TYPE "C501_VAR_TME_TYPIC"
   STRUCT
      MWA { ExternalAccessible := 'False'; ExternalVisible := 'False'; ExternalWritable := 'False'} : USInt;   // Meetwaarde
      OBS { ExternalAccessible := 'False'; ExternalVisible := 'False'; ExternalWritable := 'False'} : USInt;   // Observeerbaarheid
   END_STRUCT;
END_TYPE

TYPE "C501_VAR_TRA_TYPIC"
   STRUCT
      OBS { ExternalAccessible := 'False'; ExternalVisible := 'False'; ExternalWritable := 'False'} : USInt;   // Observeerbaarheid
   END_STRUCT;
END_TYPE

TYPE "C904_STU_IF_DEB_TYPIC"
   STRUCT
      DEB_MWA { ExternalAccessible := 'False'; ExternalVisible := 'False'; ExternalWritable := 'False'} : Real;   // Meetwaarde
      EXT_AUT { ExternalAccessible := 'False'; ExternalVisible := 'False'; ExternalWritable := 'False'} : Bool;   // Externe (hoofd) beveiliging aangesproken
      EXT_HW { ExternalAccessible := 'False'; ExternalVisible := 'False'; ExternalWritable := 'False'} : Bool;   // Sturings hardware (PLC) in storing
      STO { ExternalAccessible := 'False'; ExternalVisible := 'False'; ExternalWritable := 'False'} : Struct   // Opsomming van alle storingen
         "a" : Bool;
      END_STRUCT;
   END_STRUCT;
END_TYPE

TYPE "C904_STU_IF_NIV_TYPIC"
   STRUCT
      NIV_MWA { ExternalAccessible := 'False'; ExternalVisible := 'False'; ExternalWritable := 'False'} : Real;   // Meetwaarde
      LW { ExternalAccessible := 'False'; ExternalVisible := 'False'; ExternalWritable := 'False'} : USInt;   // Stoppeil alle pompen
      SW { ExternalAccessible := 'False'; ExternalVisible := 'False'; ExternalWritable := 'False'} : USInt;   // Startpeil pomp 1 in regime leeghouden en lozen
      MSW { ExternalAccessible := 'False'; ExternalVisible := 'False'; ExternalWritable := 'False'} : USInt;   // Startpeil pomp 2 in regime leeghouden
      LHW { ExternalAccessible := 'False'; ExternalVisible := 'False'; ExternalWritable := 'False'} : USInt;   // Stoppeil bij regime Bergen
      HHW { ExternalAccessible := 'False'; ExternalVisible := 'False'; ExternalWritable := 'False'} : USInt;   // startpeil alle pompen bij regime Bergen
      EXT_AUT { ExternalAccessible := 'False'; ExternalVisible := 'False'; ExternalWritable := 'False'} : Bool;   // Externe (hoofd) beveiliging aangesproken
      EXT_HW { ExternalAccessible := 'False'; ExternalVisible := 'False'; ExternalWritable := 'False'} : Bool;   // Sturings hardware (PLC) in storing
      STO { ExternalAccessible := 'False'; ExternalVisible := 'False'; ExternalWritable := 'False'} : Struct   // Opsomming van alle storingen
         "a" : Bool;
      END_STRUCT;
   END_STRUCT;
END_TYPE

TYPE "C904_STU_IF_PMP_TYPIC"
   STRUCT
      CMD { ExternalAccessible := 'False'; ExternalVisible := 'False'; ExternalWritable := 'False'} : Bool;   // Aansturing pomp (TRUE = AAN / FALSE = UIT)
      CMD_RES { ExternalAccessible := 'False'; ExternalVisible := 'False'; ExternalWritable := 'False'} : Bool;   // Reset van de latched storingen
   END_STRUCT;
END_TYPE

TYPE "C904_VAR_DEB_TYPIC"
   STRUCT
      MWA { ExternalAccessible := 'False'; ExternalVisible := 'False'; ExternalWritable := 'False'} : USInt;   // Meetwaarde
      OBS { ExternalAccessible := 'False'; ExternalVisible := 'False'; ExternalWritable := 'False'} : USInt;   // Observeerbaarheid
   END_STRUCT;
END_TYPE

TYPE "C904_VAR_IF_PMP_TYPIC"
   STRUCT
      STS_AAN { ExternalAccessible := 'False'; ExternalVisible := 'False'; ExternalWritable := 'False'} : Bool;   // Pomp draait
      BMO_HAND { ExternalAccessible := 'False'; ExternalVisible := 'False'; ExternalWritable := 'False'} : Bool;   // Pomp in hand geschakeld
      TYD_TOT_AAN { ExternalAccessible := 'False'; ExternalVisible := 'False'; ExternalWritable := 'False'} : LInt;   // Totaal aantal draaiuren
      TYD_TOT_AAN_UUR { ExternalAccessible := 'False'; ExternalVisible := 'False'; ExternalWritable := 'False'} : LInt;   // Totaal aantal draaiuren
      TYD_AAN { ExternalAccessible := 'False'; ExternalVisible := 'False'; ExternalWritable := 'False'} : Int;   // Aantal seconden dat pomp aangeschakeld is
      TYD_UIT { ExternalAccessible := 'False'; ExternalVisible := 'False'; ExternalWritable := 'False'} : Int;   // Aantal seconden dat pomp uitgeschakeld is
      ENE_MWA1 { ExternalAccessible := 'False'; ExternalVisible := 'False'; ExternalWritable := 'False'} : Real;   // Stroommeting fase 1
      ENE_MWA2 { ExternalAccessible := 'False'; ExternalVisible := 'False'; ExternalWritable := 'False'} : Real;   // Stroommeting fase 2
      ENE_MWA3 { ExternalAccessible := 'False'; ExternalVisible := 'False'; ExternalWritable := 'False'} : Real;   // Stroommeting fase 3
      EXT_AUT { ExternalAccessible := 'False'; ExternalVisible := 'False'; ExternalWritable := 'False'} : Bool;   // Externe (hoofd) beveiliging aangesproken
      EXT_HW { ExternalAccessible := 'False'; ExternalVisible := 'False'; ExternalWritable := 'False'} : Bool;   // Sturings hardware (PLC) in storing
      STO { ExternalAccessible := 'False'; ExternalVisible := 'False'; ExternalWritable := 'False'} : Struct   // Opsomming van alle storingen
         A001 : Bool;   // Beveiliging aangesproken
         A002 : Bool;   // Storing van de motorbeveiliging van de pomp
         A003 : Bool;   // Storing motorlade
         A004 : Bool;   // Te hoge temperatuur in de motorwikkelingen
         A005 : Bool;   // Fout stroommeting fase 1
         A006 : Bool;   // Fout stroommeting fase 2
         A007 : Bool;   // Fout stroommeting fase 3
         A008 : Bool;   // Droogloop beveiliging actief: LLW vlotter bovenwater
         A009 : Bool;   // Lekdetectie pomp
         A010 : Bool;   // Motorlade uitgeschakeld
         A011 : Bool;   // Motorlade in test
         A012 : Bool;   // Motorlade uitgereden
         AT01 : Bool;   // Discordantie motor: terugmelding niet ontvangen
         AT02 : Bool;   // Discordantie motor: terugmelding blijft aanwezig
         M001 : Bool;   // Werkschakelaar uitgeschakeld
         M002 : Bool;   // Melding: Pomp heeft te lang niet gedraaid. Periodiek onderhoud nodig
      END_STRUCT;
   END_STRUCT;
END_TYPE

TYPE "C904_VAR_IF_SPI_TYPIC"
   STRUCT
      WRE { ExternalAccessible := 'False'; ExternalVisible := 'False'; ExternalWritable := 'False'} : USInt;   // Actueel actief regime
      BMO_HAND { ExternalAccessible := 'False'; ExternalVisible := 'False'; ExternalWritable := 'False'} : Bool;   // TRUE = Regime handmatig ingesteld via lokale bediening
      STO { ExternalAccessible := 'False'; ExternalVisible := 'False'; ExternalWritable := 'False'} : Struct   // Opsomming van alle storingen
         A001 : Bool;   // Beveiliging aangesproken
         A002 : Bool;   // Beveiliging No-Break aangesproken
         A003 : Bool;   // Overspanningsbeveiliging aangesproken
         A004 : Bool;   // Schuif ALSB uitgeschakeld
         A005 : Bool;   // Schuif ALSB in test
         A006 : Bool;   // Schuif ALSB uitgereden
         A007 : Bool;   // Nisdeur niet gesloten
         A008 : Bool;   // Storing tracing
      END_STRUCT;
   END_STRUCT;
END_TYPE

TYPE "C904_VAR_IF_VPI_TYPIC"
   STRUCT
      WRE { ExternalAccessible := 'False'; ExternalVisible := 'False'; ExternalWritable := 'False'} : USInt;   // Actueel actief regime
      BMO_HAND { ExternalAccessible := 'False'; ExternalVisible := 'False'; ExternalWritable := 'False'} : Bool;   // TRUE = Regime handmatig ingesteld via lokale bediening
   END_STRUCT;
END_TYPE

TYPE "C904_VAR_NIV_TYPIC"
   STRUCT
      MWA { ExternalAccessible := 'False'; ExternalVisible := 'False'; ExternalWritable := 'False'} : USInt;   // Meetwaarde
      STS_LW { ExternalAccessible := 'False'; ExternalVisible := 'False'; ExternalWritable := 'False'} : USInt;   // Stoppeil alle pompen
      STS_SW { ExternalAccessible := 'False'; ExternalVisible := 'False'; ExternalWritable := 'False'} : USInt;   // Startpeil pomp 1 in regime leeghouden en lozen
      STS_MSW { ExternalAccessible := 'False'; ExternalVisible := 'False'; ExternalWritable := 'False'} : USInt;   // Startpeil pomp 2 in regime leeghouden
      STS_LHW { ExternalAccessible := 'False'; ExternalVisible := 'False'; ExternalWritable := 'False'} : USInt;   // Stoppeil bij regime Bergen
      STS_HHW { ExternalAccessible := 'False'; ExternalVisible := 'False'; ExternalWritable := 'False'} : USInt;   // Startpeil alle pompen bij regime Bergen
      OBS { ExternalAccessible := 'False'; ExternalVisible := 'False'; ExternalWritable := 'False'} : USInt;   // Observeerbaarheid
   END_STRUCT;
END_TYPE

TYPE "C904_VAR_PMP_TYPIC"
   STRUCT
      STS { ExternalAccessible := 'False'; ExternalVisible := 'False'; ExternalWritable := 'False'} : USInt;   // Status van de pomp
      BMO { ExternalAccessible := 'False'; ExternalVisible := 'False'; ExternalWritable := 'False'} : USInt;   // Bedieningsmode
      BST { ExternalAccessible := 'False'; ExternalVisible := 'False'; ExternalWritable := 'False'} : USInt;   // Bestuurbaarheid
      LLW { ExternalAccessible := 'False'; ExternalVisible := 'False'; ExternalWritable := 'False'} : USInt;   // Vlotter droogloopbewaking
      PWR { ExternalAccessible := 'False'; ExternalVisible := 'False'; ExternalWritable := 'False'} : Real;   // Actueel vermogen van de pomp
      TYD_TOT_AAN { ExternalAccessible := 'False'; ExternalVisible := 'False'; ExternalWritable := 'False'} : USInt;   // Totaal aantal draaiuren
      TYD_AAN { ExternalAccessible := 'False'; ExternalVisible := 'False'; ExternalWritable := 'False'} : USInt;   // Tijdsduur dat pomp aangeschakeld is
      TYD_UIT { ExternalAccessible := 'False'; ExternalVisible := 'False'; ExternalWritable := 'False'} : USInt;   // Tijdsduur dat pomp uitgeschakeld is
   END_STRUCT;
END_TYPE

TYPE "C215_STU_IF_DVLU_TYPIC"
   STRUCT
      CMD_OPL { ExternalAccessible := 'False'; ExternalVisible := 'False'; ExternalWritable := 'False'} : Bool;   // Aansturing indicatiebord vluchtroute oplopende richting
      CMD_AFL { ExternalAccessible := 'False'; ExternalVisible := 'False'; ExternalWritable := 'False'} : Bool;   // Aansturing indicatiebord vluchtroute aflopende richting
      CMD_RES { ExternalAccessible := 'False'; ExternalVisible := 'False'; ExternalWritable := 'False'} : Bool;   // Reset van de latched storingen
   END_STRUCT;
END_TYPE

TYPE "C215_STU_IF_SVLU_TYPIC"
   STRUCT
      CMD_AAN { ExternalAccessible := 'False'; ExternalVisible := 'False'; ExternalWritable := 'False'} : Bool;   // Aansturing statisch indicatiebord vluchtroute
      CMD_RES { ExternalAccessible := 'False'; ExternalVisible := 'False'; ExternalWritable := 'False'} : Bool;   // Reset van de latched storingen
   END_STRUCT;
END_TYPE

TYPE "C215_VAR_DVLU_TYPIC"
   STRUCT
      STS { ExternalAccessible := 'False'; ExternalVisible := 'False'; ExternalWritable := 'False'} : USInt;   // Status van het dynamisch indicatiebord vluchtroute
      BST { ExternalAccessible := 'False'; ExternalVisible := 'False'; ExternalWritable := 'False'} : USInt;   // Bestuurbaarheid
   END_STRUCT;
END_TYPE

TYPE "C215_VAR_IF_DVLU_TYPIC"
   STRUCT
      STS_OPL { ExternalAccessible := 'False'; ExternalVisible := 'False'; ExternalWritable := 'False'} : Bool;   // Indicatiebord vluchtroute aangestuurd in oplopende richting
      STS_AFL { ExternalAccessible := 'False'; ExternalVisible := 'False'; ExternalWritable := 'False'} : Bool;   // Indicatiebord vluchtroute aangestuurd in aflopende richting
      EXT_AUT { ExternalAccessible := 'False'; ExternalVisible := 'False'; ExternalWritable := 'False'} : Bool;   // Externe (hoofd) beveiliging aangesproken
      EXT_HW { ExternalAccessible := 'False'; ExternalVisible := 'False'; ExternalWritable := 'False'} : Bool;   // Sturings hardware (PLC) in storing
      STO { ExternalAccessible := 'False'; ExternalVisible := 'False'; ExternalWritable := 'False'} : Struct   // Opsomming van alle storingen
         A001 : Bool;   // Beveiliging aangesproken
         AT01 : Bool;   // Foute terugmelding: Indicatiebord uitgestuurd, terugmelding Uit niet (of te laat) ontvangen
         AT02 : Bool;   // Foute terugmelding: Indicatiebord niet uitgestuurd, terugmelding Uit blijft aanwezig
         AT03 : Bool;   // Foute terugmelding: Oplopend aangestuurd, terugmelding Aan niet (of te laat) ontvangen
         AT04 : Bool;   // Foute terugmelding: Oplopend niet aangestuurd, terugmelding Aan blijft aanwezig
         AT05 : Bool;   // Foute terugmelding: Aflopend aangestuurd, terugmelding Aan niet (of te laat) ontvangen
         AT06 : Bool;   // Foute terugmelding: Aflopend niet aangestuurd, terugmelding Aan blijft aanwezig
         AT07 : Bool;   // Foute terugmeldingen: terugmeldingen oplopend en aflopend tegelijkertijd
      END_STRUCT;
   END_STRUCT;
END_TYPE

TYPE "C215_VAR_IF_PBK_TYPIC"
   STRUCT
      EXT_AUT { ExternalAccessible := 'False'; ExternalVisible := 'False'; ExternalWritable := 'False'} : Bool;   // Externe (hoofd) beveiliging aangesproken
      EXT_HW { ExternalAccessible := 'False'; ExternalVisible := 'False'; ExternalWritable := 'False'} : Bool;   // Sturings hardware (PLC) in storing
      STO { ExternalAccessible := 'False'; ExternalVisible := 'False'; ExternalWritable := 'False'} : Struct   // Opsomming van alle storingen
         A001 : Bool;   // Beveiliging aangesproken
         A002 : Bool;   // Storing batterij
      END_STRUCT;
   END_STRUCT;
END_TYPE

TYPE "C215_VAR_IF_SVLU_TYPIC"
   STRUCT
      STS_UIT { ExternalAccessible := 'False'; ExternalVisible := 'False'; ExternalWritable := 'False'} : Bool;   // Statisch indicatiebord vluchtroute uit
      EXT_AUT { ExternalAccessible := 'False'; ExternalVisible := 'False'; ExternalWritable := 'False'} : Bool;   // Externe (hoofd) beveiliging aangesproken
      EXT_HW { ExternalAccessible := 'False'; ExternalVisible := 'False'; ExternalWritable := 'False'} : Bool;   // Sturings hardware (PLC) in storing
      STO { ExternalAccessible := 'False'; ExternalVisible := 'False'; ExternalWritable := 'False'} : Struct   // Opsomming van alle storingen
         A001 : Bool;   // Beveiliging aangesproken
         AT01 : Bool;   // Foute terugmelding: Indicatiebord uitgestuurd, terugmelding Uit niet (of te laat) ontvangen
         AT02 : Bool;   // Foute terugmelding: Indicatiebord niet uitgestuurd, terugmelding Uit blijft aanwezig
      END_STRUCT;
   END_STRUCT;
END_TYPE

TYPE "C215_VAR_SVLU_TYPIC"
   STRUCT
      STS { ExternalAccessible := 'False'; ExternalVisible := 'False'; ExternalWritable := 'False'} : USInt;   // Status van het statisch indicatiebord vluchtroute
      BST { ExternalAccessible := 'False'; ExternalVisible := 'False'; ExternalWritable := 'False'} : USInt;   // Bestuurbaarheid
   END_STRUCT;
END_TYPE

ORGANIZATION_BLOCK "Main"   // OB1, LAD, ProgramCycle
TITLE = "Main Program Sweep (Cycle)"
{ S7_Optimized_Access := 'TRUE' }
// stored: SetENOAutomatically false
   VAR_INPUT
      Initial_Call : Bool;   // Initial call of this OB
      Remanence : Bool;   // =True, if remanent data are available
   END_VAR
BEGIN
END_ORGANIZATION_BLOCK

FUNCTION_BLOCK "TYPIC_C701_IF_KLB"   // FB120, FBD
TITLE = TYPIC_C701_IF_KLB: Brandklep
{ S7_Optimized_Access := 'TRUE' }
AUTHOR : OCOTECH
FAMILY : Typical
NAME : C701.708
// Logisch Object Besturing: C701.708
// 
// De interne functie Brandklep verzorgt de interne besturing, bewaking en fysieke aansturing van een brandklep.
// stored: MemoryReserve 10, SetENOAutomatically false
   VAR_INPUT
      IN_KLB { ExternalAccessible := 'False'; ExternalVisible := 'False'; ExternalWritable := 'False'} : Bool;   // Status brandklep (1 = Open)
   END_VAR
   VAR_OUTPUT
      VAR_IF_KLB { ExternalAccessible := 'False'; ExternalVisible := 'False'; ExternalWritable := 'False'} : "C701_VAR_IF_KLB_TYPIC";   // Struct met alle variabelen naar bovenliggende functies
   END_VAR
   VAR
      STO { ExternalWritable := 'False'} : Struct   // Storingen
         A001 : Bool;   // Brandklep gesloten
      END_STRUCT;
      VAR { ExternalWritable := 'False'} : Struct   // Variabelen
         KLB_TOE { ExternalAccessible := 'False'; ExternalVisible := 'False'} : Bool;   // Brandklep gesloten
      END_STRUCT;
   END_VAR
BEGIN

REGION Network 1: START
END_REGION

REGION Network 2: +++ Storingen +++
   // aanmaken storingen.
END_REGION

REGION Network 3: Storing A001: Brandklep gesloten
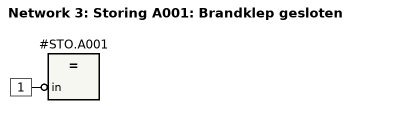
   #STO.A001 := NOT 1;
END_REGION

REGION Network 4 (SCL): EINDE
   // Variabelen van intern scada rakvlak naar outputs copieren
   #VAR_IF_KLB.KLB_TOE := #VAR.KLB_TOE;
END_REGION
END_FUNCTION_BLOCK

FUNCTION_BLOCK "TYPIC_C701_IF_KMO"   // FB102, FBD
TITLE = TYPIC_C701_IF_KMO: Koelmachine
{ S7_Optimized_Access := 'TRUE' }
AUTHOR : OCOTECH
FAMILY : Typical
NAME : C701.715
// Logisch Object Besturing: C701.715
// 
// De interne functie koelmachine verzorgt de interne besturing, bewaking en fysieke aansturing van de koelmachine behorend tot de klimaatinstallatie.
// stored: MemoryReserve 10, SetENOAutomatically false
   VAR_INPUT
      STU_IF_KMO { ExternalAccessible := 'False'; ExternalVisible := 'False'; ExternalWritable := 'False'} : Bool;   // Sturing van de interne functie klimaatregeling (IF), koudevraag voor kring
      IN_TME_IN { ExternalAccessible := 'False'; ExternalVisible := 'False'; ExternalWritable := 'False'} : Real;   // Temperatuurmeting koud water in
      IN_TME_UIT { ExternalAccessible := 'False'; ExternalVisible := 'False'; ExternalWritable := 'False'} : Real;   // Temperatuurmeting koud water uit
      IN_DME { ExternalAccessible := 'False'; ExternalVisible := 'False'; ExternalWritable := 'False'} : Real;   // Drukmeting koelen
      IN_SCF { ExternalAccessible := 'False'; ExternalVisible := 'False'; ExternalWritable := 'False'} : Bool;   // Flowmeting (1 = Flow)
      IN_FB_VGV { ExternalAccessible := 'False'; ExternalVisible := 'False'; ExternalWritable := 'False'} : Bool;   // Feedback sturing vrijgave (1 = Vrijgave)
      IN_AL { ExternalAccessible := 'False'; ExternalVisible := 'False'; ExternalWritable := 'False'} : Bool;   // Algemeen alarm koelmachine (1 = Alarm)
      IN_PMP { ExternalAccessible := 'False'; ExternalVisible := 'False'; ExternalWritable := 'False'} : Bool;   // Status circulatiepomp (1 = Aan)
      IN_AL_PMP { ExternalAccessible := 'False'; ExternalVisible := 'False'; ExternalWritable := 'False'} : Bool;   // Storing circulatiepomp (1 = Storing)
      IN_KLP { ExternalAccessible := 'False'; ExternalVisible := 'False'; ExternalWritable := 'False'} : Bool;   // Status klep (1 = Open)
   END_VAR
   VAR_OUTPUT
      VAR_IF_KMO { ExternalAccessible := 'False'; ExternalVisible := 'False'; ExternalWritable := 'False'} : "C701_VAR_IF_KMO_TYPIC";   // Struct met alle variabelen naar bovenliggende functies
      OUT_VGV { ExternalAccessible := 'False'; ExternalVisible := 'False'; ExternalWritable := 'False'} : Bool;   // Vrijgave koelmachine
      OUT_SWA_TME { ExternalAccessible := 'False'; ExternalVisible := 'False'; ExternalWritable := 'False'} : Real;   // Setpunt temperatuur koelwater
      OUT_KLP { ExternalAccessible := 'False'; ExternalVisible := 'False'; ExternalWritable := 'False'} : Bool;   // Aansturing 2wegklep
   END_VAR
   VAR
      STO { ExternalWritable := 'False'} : Struct   // Storingen
         A001 : Bool;   // Fout temperatuurmeting koelwater in
         A002 : Bool;   // Fout temperatuurmeting koelwater uit
         A003 : Bool;   // Fout drukmeting koelwater
         A004 : Bool;   // Fout flowmeting koelwater
         A005 : Bool;   // Fout algemeen koelmachine
         A006 : Bool;   // Fout circulatiepomp
      END_STRUCT;
      VAR { ExternalWritable := 'False'} : Struct   // Variabelen
         TME_IN : Real;   // Temperatuurmeting koelwater in
         TME_UIT : Real;   // Temperatuurmeting koelwater uit
         DME : Real;   // Drukmeting koelwater
         SWA_TME : Real;   // Setpunt koelwater
      END_STRUCT;
   END_VAR
BEGIN

REGION Network 1: START
END_REGION

REGION Network 2: +++ Metingen +++
   // inlezen van temperaturen en druk.
END_REGION

REGION Network 3: +++ Storingen en meldingen +++
   // aanmaken van storingen en meldingen.
END_REGION

REGION Network 4: Storing A001: Fout temperatuurmeting koelwater in
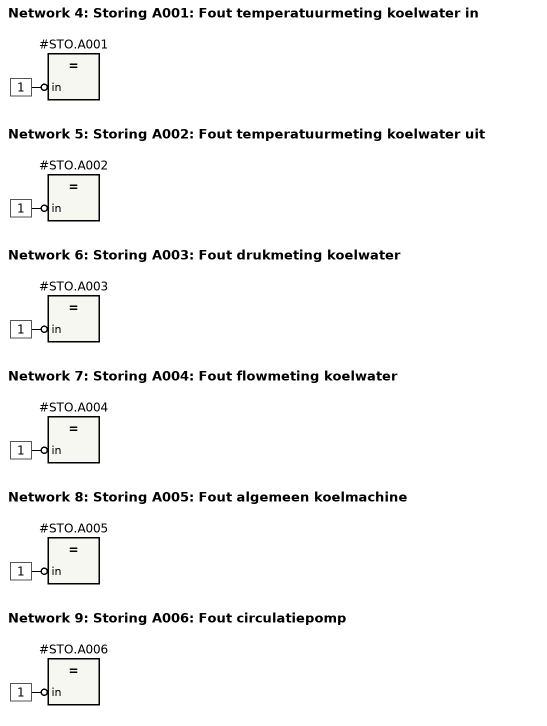
   #STO.A001 := NOT 1;
END_REGION

REGION Network 5: Storing A002: Fout temperatuurmeting koelwater uit
   #STO.A002 := NOT 1;
END_REGION

REGION Network 6: Storing A003: Fout drukmeting koelwater
   #STO.A003 := NOT 1;
END_REGION

REGION Network 7: Storing A004: Fout flowmeting koelwater
   #STO.A004 := NOT 1;
END_REGION

REGION Network 8: Storing A005: Fout algemeen koelmachine
   #STO.A005 := NOT 1;
END_REGION

REGION Network 9: Storing A006: Fout circulatiepomp
   #STO.A006 := NOT 1;
END_REGION

REGION Network 10: +++ Sturingen +++
   // sturing van klep en vrijgave koelmachine in functie van koelvraag.
END_REGION

REGION Network 11 (SCL): EINDE
   // Variabelen van intern scada rakvlak naar outputs copieren
   #VAR_IF_KMO.STO := #STO;
END_REGION
END_FUNCTION_BLOCK

FUNCTION_BLOCK "TYPIC_C701_IF_KOKR"   // FB101, FBD
TITLE = TYPIC_C701_IF_KOKR: Koelkring
{ S7_Optimized_Access := 'TRUE' }
AUTHOR : OCOTECH
FAMILY : Typical
NAME : C701.712
// Logisch Object Besturing: C701.712
// 
// De interne functie Koelkring verzorgt de interne besturing, bewaking en fysieke aansturing van een kring van de collector behorend tot de klimaatinstallatie.
// Er wordt een vrijgave aan de pompen gegeven als er een koelvraag is. De drukregeling gebeurt door de pomp zelf. Antioblokkeer beveiliging is ook instelbaar op de pomp zelf.
// Indien er een tweede pomp is, wordt deze afwisselend gebruikt. Of wordt er gewisseld bij een storing van de actieve pomp.
// De collector koelkring bestaat uit 2 kringen:
//  Kring ventiloconvectoren en klimaatkasten
//  Kring koelbatterij luchtgroep
// stored: MemoryReserve 10, SetENOAutomatically false
   VAR_INPUT
      STU_IF_KOKR { ExternalAccessible := 'False'; ExternalVisible := 'False'; ExternalWritable := 'False'} : Bool;   // Sturing van de interne functie klimaatregeling (IF), koudevraag voor kring
      IN_AAN_PMP1 { ExternalAccessible := 'False'; ExternalVisible := 'False'; ExternalWritable := 'False'} : Bool;   // Terugmelding aansturing pomp 1 (1 = Aan)
      IN_AAN_PMP2 { ExternalAccessible := 'False'; ExternalVisible := 'False'; ExternalWritable := 'False'} : Bool;   // Terugmelding aansturing pomp 2 (1 = Aan)
      IN_THM_PMP1 { ExternalAccessible := 'False'; ExternalVisible := 'False'; ExternalWritable := 'False'} : Bool;   // Status thermische beveiliging (1 = OK) pomp 1
      IN_THM_PMP2 { ExternalAccessible := 'False'; ExternalVisible := 'False'; ExternalWritable := 'False'} : Bool;   // Status thermische beveiliging (1 = OK) pomp 2
      IN_DME { ExternalAccessible := 'False'; ExternalVisible := 'False'; ExternalWritable := 'False'} : Real;   // Drukmeting
      IN_TME_IN { ExternalAccessible := 'False'; ExternalVisible := 'False'; ExternalWritable := 'False'} : Real;   // Temperatuur vertrek
      IN_TME_UIT { ExternalAccessible := 'False'; ExternalVisible := 'False'; ExternalWritable := 'False'} : Real;   // Temperatuur retour
      CFG_TYD_FB { ExternalAccessible := 'False'; ExternalVisible := 'False'; ExternalWritable := 'False'} : Time;   // Vertragingstijd storing foute terugmelding
      CFG_PMP { ExternalAccessible := 'False'; ExternalVisible := 'False'; ExternalWritable := 'False'} : Bool;   // True = Kring met 2 pompen
      CFG_PMP_TYD { ExternalAccessible := 'False'; ExternalVisible := 'False'; ExternalWritable := 'False'} : Time;   // Maximale draaitijd voor wisselen pomp
   END_VAR
   VAR_OUTPUT
      VAR_IF_KOKR { ExternalAccessible := 'False'; ExternalVisible := 'False'; ExternalWritable := 'False'} : "C701_VAR_IF_KOKR_TYPIC";   // Struct met alle variabelen naar bovenliggende functies
      OUT_VGV_PMP1 { ExternalAccessible := 'False'; ExternalVisible := 'False'; ExternalWritable := 'False'} : Bool;   // Vrijgave pomp 1
      OUT_VGV_PMP2 { ExternalAccessible := 'False'; ExternalVisible := 'False'; ExternalWritable := 'False'} : Bool;   // Vrijgave pomp 2
   END_VAR
   VAR_IN_OUT
      STU_VGV_KOKR_AAN : Bool;   // Vrijgave inschakelen NIET NODIG?
   END_VAR
   VAR
      STO { ExternalWritable := 'False'} : Struct   // Storingen
         A001 : Bool;   // Storing van de motorbeveiliging van pomp 1
         A002 : Bool;   // Storing van de motorbeveiliging van pomp 2
         A003 : Bool;   // Fout temperatuurmeting vertrek
         A004 : Bool;   // Fout temperatuurmeting retour
         A005 : Bool;   // Fout drukmeting
      END_STRUCT;
      VAR { ExternalWritable := 'False'} : Struct   // Variabelen
         TME_IN : Real;   // Temperatuur vertrek
         TME_UIT : Real;   // Temperatuur retour
         DME : Real;   // Druk vertrek
         VGV_P1 : Bool;   // Vrijgave voor pomp 1
         VGV_P2 : Bool;   // Vrijgave voor pomp 2
         TYD_TOT_AAN_P1 : LInt;   // Totaal aantal draaiuren (in seconden)
         TYD_TOT_AAN_UUR_P1 : LInt;   // Totaal aantal draaiuren (in uren)
         TYD_TOT_AAN_P2 : LInt;   // Totaal aantal draaiuren (in seconden)
         TYD_TOT_AAN_UUR_P2 : LInt;   // Totaal aantal draaiuren (in uren)
         TYD_AAN_P1 : LInt;   // Aantal seconden dat pomp aangeschakeld is
         TYD_AAN_P2 : LInt;   // Aantal seconden dat pomp aangeschakeld is
      END_STRUCT;
   END_VAR
BEGIN

REGION Network 1: START
END_REGION

REGION Network 2: +++ Metingen +++
   // inlezen van vertrek- en retourtemperatuur.
END_REGION

REGION Network 3: +++ Storingen en meldingen +++
   // aanmaken van storingen en meldingen.
END_REGION

REGION Network 4: Storing A001: Storing van de motorbeveiliging van pomp 1
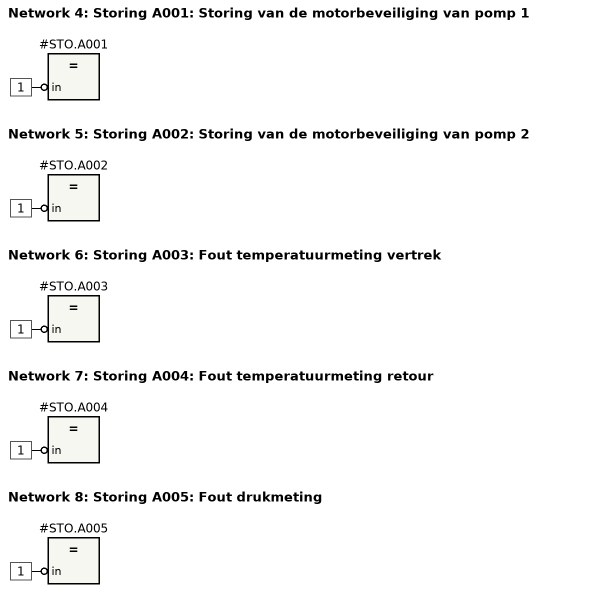
   #STO.A001 := NOT 1;
END_REGION

REGION Network 5: Storing A002: Storing van de motorbeveiliging van pomp 2
   #STO.A002 := NOT 1;
END_REGION

REGION Network 6: Storing A003: Fout temperatuurmeting vertrek
   #STO.A003 := NOT 1;
END_REGION

REGION Network 7: Storing A004: Fout temperatuurmeting retour
   #STO.A004 := NOT 1;
END_REGION

REGION Network 8: Storing A005: Fout drukmeting
   #STO.A005 := NOT 1;
END_REGION

REGION Network 9: +++ Sturingen pomp +++
   // bij koudevraag pomp vrijgave geven.
END_REGION

REGION Network 10: +++ Urentellers +++
   // tellen van de tijdsduur dat de motor draait.
END_REGION

REGION Network 11 (SCL): EINDE
   // Variabelen van intern scada rakvlak naar outputs copieren
   #VAR_IF_KOKR.STO := #STO;
END_REGION
END_FUNCTION_BLOCK

FUNCTION_BLOCK "TYPIC_C701_IF_LBS"   // FB83, FBD
TITLE = TYPIC_C701_IF_LBS: Luchtbehandelingssysteem
{ S7_Optimized_Access := 'TRUE' }
AUTHOR : OCOTECH
FAMILY : Typical
NAME : C701.702
// Logisch Object Besturing: C701.702
// 
// De interne functie Luchtbehandelingssysteem verzorgt de interne besturing, bewaking en fysieke aansturing van de luchtgroep behorend tot de klimaatinstallatie.
// stored: MemoryReserve 10, SetENOAutomatically false
   VAR_INPUT
      STU_IF_LBS_CMD { ExternalAccessible := 'False'; ExternalVisible := 'False'; ExternalWritable := 'False'} : USInt;   // Sturing van de interne functie klimaatregeling (IF), luchtgroep
      IN_DME_PU { ExternalAccessible := 'False'; ExternalVisible := 'False'; ExternalWritable := 'False'} : Real;   // Drukmeting in pulsie kanaal
      IN_DME_EX { ExternalAccessible := 'False'; ExternalVisible := 'False'; ExternalWritable := 'False'} : Real;   // Drukmeting in extractie kanaal
      IN_TME_PU { ExternalAccessible := 'False'; ExternalVisible := 'False'; ExternalWritable := 'False'} : Real;   // Temperatuurmeting in pulsie kanaal
      IN_TME_EX { ExternalAccessible := 'False'; ExternalVisible := 'False'; ExternalWritable := 'False'} : Real;   // Temperatuurmeting in extractie kanaal
      IN_TME_BU { ExternalAccessible := 'False'; ExternalVisible := 'False'; ExternalWritable := 'False'} : Real;   // Temperatuurmeting buiten
      IN_VEN_PU { ExternalAccessible := 'False'; ExternalVisible := 'False'; ExternalWritable := 'False'} : Bool;   // Status pulsie ventilator (on/off)
      IN_VEN_PU_FB { ExternalAccessible := 'False'; ExternalVisible := 'False'; ExternalWritable := 'False'} : Real;   // Feedback snelheid pulsie ventilator
      IN_VEN_PU_AUT { ExternalAccessible := 'False'; ExternalVisible := 'False'; ExternalWritable := 'False'} : Bool;   // Status thermische beveiliging pulsie ventilator (1 = OK)
      IN_VEN_PU_SCW { ExternalAccessible := 'False'; ExternalVisible := 'False'; ExternalWritable := 'False'} : Bool;   // Werkschakelaar pulsie ventilator (1 = Aan)
      IN_VEN_EX { ExternalAccessible := 'False'; ExternalVisible := 'False'; ExternalWritable := 'False'} : Bool;   // Status extractie ventilator (on/off)
      IN_VEN_EX_FB { ExternalAccessible := 'False'; ExternalVisible := 'False'; ExternalWritable := 'False'} : Real;   // Feedback snelheid extractie ventilator
      IN_VEN_EX_AUT { ExternalAccessible := 'False'; ExternalVisible := 'False'; ExternalWritable := 'False'} : Bool;   // Status thermische beveiliging extractie ventilator (1 = OK)
      IN_VEN_EX_SCW { ExternalAccessible := 'False'; ExternalVisible := 'False'; ExternalWritable := 'False'} : Bool;   // Werkschakelaar extractie ventilator (1 = Aan)
      IN_KLR_KOB { ExternalAccessible := 'False'; ExternalVisible := 'False'; ExternalWritable := 'False'} : Real;   // Feedback stand 2weg klep koelbatterij
      IN_KLR_VEB { ExternalAccessible := 'False'; ExternalVisible := 'False'; ExternalWritable := 'False'} : Real;   // Feedback stand 3weg klep verwarmingsbatterij
      IN_KLR_PU { ExternalAccessible := 'False'; ExternalVisible := 'False'; ExternalWritable := 'False'} : Real;   // Terugmelding stand open/dicht register verse lucht
      IN_KLR_EX { ExternalAccessible := 'False'; ExternalVisible := 'False'; ExternalWritable := 'False'} : Real;   // Terugmelding stand open/dicht register extractie
      IN_KLR { ExternalAccessible := 'False'; ExternalVisible := 'False'; ExternalWritable := 'False'} : Real;   // Terugmelding stand mengregister
      IN_AVR { ExternalAccessible := 'False'; ExternalVisible := 'False'; ExternalWritable := 'False'} : Bool;   // Antivries schakelaar (1 = OK)
      IN_DME_FI_VL { ExternalAccessible := 'False'; ExternalVisible := 'False'; ExternalWritable := 'False'} : Bool;   // Drukverschilmeting filter verse lucht (1 = OK)
      IN_DME_FI_EX { ExternalAccessible := 'False'; ExternalVisible := 'False'; ExternalWritable := 'False'} : Bool;   // Drukverschilmeting filter extractie (1 = OK)
      IN_WMW { ExternalAccessible := 'False'; ExternalVisible := 'False'; ExternalWritable := 'False'} : Bool;   // Terugmelding status warmtewiel (Aan / Uit)
      IN_WMW_STO { ExternalAccessible := 'False'; ExternalVisible := 'False'; ExternalWritable := 'False'} : Bool;   // Fout warmtewiel (1 = OK)
      IN_BME { ExternalAccessible := 'False'; ExternalVisible := 'False'; ExternalWritable := 'False'} : Bool;   // Rookmelder (1 = OK)
      CFG_TYD_FB { ExternalAccessible := 'False'; ExternalVisible := 'False'; ExternalWritable := 'False'} : Time;   // Vertragingstijd storing foute terugmelding
   END_VAR
   VAR_OUTPUT
      VAR_IF_LBS { ExternalAccessible := 'False'; ExternalVisible := 'False'; ExternalWritable := 'False'} : "C701_VAR_IF_LBS_TYPIC";   // Struct met alle variabelen naar bovenliggende functies
      OUT_VEN_PU_VGV { ExternalAccessible := 'False'; ExternalVisible := 'False'; ExternalWritable := 'False'} : Bool;   // Vrijgave pulsie ventilator
      OUT_VEN_PU_SNE { ExternalAccessible := 'False'; ExternalVisible := 'False'; ExternalWritable := 'False'} : Real;   // Snelheid pulsie ventilator
      OUT_VEN_EX_VGV { ExternalAccessible := 'False'; ExternalVisible := 'False'; ExternalWritable := 'False'} : Bool;   // Vrijgave extractie ventilator
      OUT_VEN_EX_SNE { ExternalAccessible := 'False'; ExternalVisible := 'False'; ExternalWritable := 'False'} : Real;   // Snelheid extractie ventilator
      OUT_KLR_KOB { ExternalAccessible := 'False'; ExternalVisible := 'False'; ExternalWritable := 'False'} : Real;   // Aansturing klep koelbatterij
      OUT_KLR_VEB { ExternalAccessible := 'False'; ExternalVisible := 'False'; ExternalWritable := 'False'} : Real;   // Aansturing klep verwarmingsbatterij
      OUT_KLR_VL { ExternalAccessible := 'False'; ExternalVisible := 'False'; ExternalWritable := 'False'} : Real;   // Damper verse lucht sturing
      OUT_KLR_EX { ExternalAccessible := 'False'; ExternalVisible := 'False'; ExternalWritable := 'False'} : Real;   // Damper extractie lucht sturing
      OUT_KLR { ExternalAccessible := 'False'; ExternalVisible := 'False'; ExternalWritable := 'False'} : Real;   // Aansturing positie mengregister
      OUT_WMW { ExternalAccessible := 'False'; ExternalVisible := 'False'; ExternalWritable := 'False'} : Real;   // Aansturing recuperatie warmtewisselaar
   END_VAR
   VAR_IN_OUT
      STU_VGV_PMP_AAN : Bool;   // Vrijgave inschakelen
   END_VAR
   VAR
      BED : Struct   // Bedieningen
         REM : Bool;   // Bediening om luchtgroep in remote te schakelen
         NORMAAL : Bool;   // Bediening om luchtgroep in regime Normaal te schakelen
         RECIRCULATIE : Bool;   // Bediening om luchtgroep in regime Recirculatie te schakelen
         UIT : Bool;   // Bediening om luchtgroep in regime Uit te schakelen
      END_STRUCT;
      STO { ExternalWritable := 'False'} : Struct   // Storingen
         A001 : Bool;   // Storing van de motorbeveiliging van pulsie ventilator
         A002 : Bool;   // Storing van de motorbeveiliging van extractie ventilator
         A003 : Bool;   // Fout drukmeting pulsie
         A004 : Bool;   // Fout drukmeting extractie
         A005 : Bool;   // Fout temperatuurmeting pulsie
         A006 : Bool;   // Fout temperatuurmeting extractie
         A007 : Bool;   // Fout temperatuurmeting buitenlucht
         A008 : Bool;   // Antivries alarm
         A009 : Bool;   // Filter vuil verse lucht
         A010 : Bool;   // Filter vuil extractie lucht
         AT01 : Bool;   // Foute terugmelding: damper verse lucht aangestuurd, terugmelding niet (of te laat) ontvangen
         AT02 : Bool;   // Foute terugmelding: damper extractie lucht aangestuurd, terugmelding niet (of te laat) ontvangen
         M001 : Bool;   // De pulsie ventilator is afgekoppeld via de werkschakelaar
         M002 : Bool;   // De extractie ventilator is afgekoppeld via de werkschakelaar
      END_STRUCT;
      VAR { ExternalWritable := 'False'} : Struct   // Variabelen
         PID_P_PU : Real;   // P factor van PID regeling voor pulsie ventilator
         PID_I_PU : Time;   // Integratietijd van PID regeling voor pulsie ventilator
         PID_D_PU : Time;   // D actie van PID regeling voor pulsie ventilator
         PID_P_EX : Real;   // P factor van PID regeling voor extractie ventilator
         PID_I_EX : Time;   // Integratietijd van PID regeling voor extractie ventilator
         PID_D_EX : Time;   // D actie van PID regeling voor extractie ventilator
         PID_P_KOB : Real;   // P factor van PID regeling voor klep van koelbatterij
         PID_I_KOB : Time;   // Integratietijd van PID regeling voor klep van koelbatterij
         PID_D_KOB : Time;   // D actie van PID regeling voor klep van koelbatterij
         PID_P_VEB : Real;   // P factor van PID regeling voor klep van verwarmingsbatterij
         PID_I_VEB : Time;   // Integratietijd van PID regeling voor klep van verwarmingsbatterij
         PID_D_VEB : Time;   // D actie van PID regeling voor klep van verwarmingsbatterij
         SWA_D_PU : Real;   // Setpunt druk pulsie kanaal
         SWA_D_EX : Real;   // Setpunt druk extractie kanaal
         SWA_T_PU : Real;   // Setpunt temperatuur pulsie
         DME_PU : Real;   // Drukmeting pulsie kanaal
         DME_EX : Real;   // Drukmeting extractie kanaal
         TME_PU : Real;   // Temperatuurmeting in pulsie
         TME_EX : Real;   // Temperatuurmeting in extractie
         TME_BU : Real;   // Temperatuurmeting buitenlucht
         WRE { ExternalAccessible := 'False'; ExternalVisible := 'False'} : USInt;   // Werkingsregime
         BMO_HAND { ExternalAccessible := 'False'; ExternalVisible := 'False'} : Bool;   // TRUE = Werkingsregime is handmatig ingesteld via lokale bediening
         "Vrijgave pomp verwarmingsbat" { ExternalAccessible := 'False'; ExternalVisible := 'False'} : Bool;   // Gaat naar if verwarmingskring CHECKEN OF DEZE POMP NU HIER INZIT OF IN DE KRING
         REQ_VE { ExternalAccessible := 'False'; ExternalVisible := 'False'} : Bool;   // Warmtevraag voor kring verwarmingsbatterijen
         REQ_KO { ExternalAccessible := 'False'; ExternalVisible := 'False'} : Bool;   // Koelvraag voor kring koelbatterijen (luchtgroep)
      END_STRUCT;
   END_VAR
BEGIN

REGION Network 1: START
END_REGION

REGION Network 2: +++ Metingen +++
   // inlezen van de temperatuur en drukken.
END_REGION

REGION Network 3: +++ Storingen en meldingen +++
   // aanmaken van de storingen en meldingen.
END_REGION

REGION Network 4: Storing A001: Storing van de motorbeveiliging van pulsie ventilator
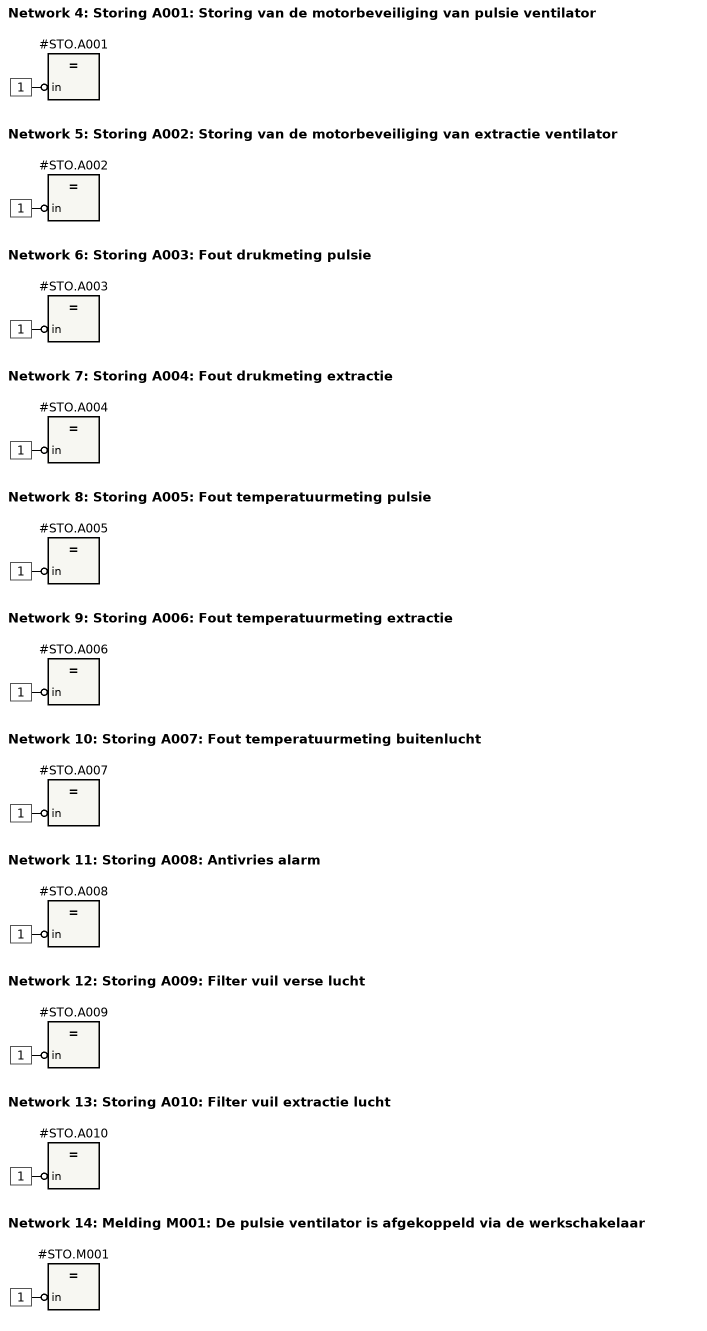
   #STO.A001 := NOT 1;
END_REGION

REGION Network 5: Storing A002: Storing van de motorbeveiliging van extractie ventilator
   #STO.A002 := NOT 1;
END_REGION

REGION Network 6: Storing A003: Fout drukmeting pulsie
   #STO.A003 := NOT 1;
END_REGION

REGION Network 7: Storing A004: Fout drukmeting extractie
   #STO.A004 := NOT 1;
END_REGION

REGION Network 8: Storing A005: Fout temperatuurmeting pulsie
   #STO.A005 := NOT 1;
END_REGION

REGION Network 9: Storing A006: Fout temperatuurmeting extractie
   #STO.A006 := NOT 1;
END_REGION

REGION Network 10: Storing A007: Fout temperatuurmeting buitenlucht
   #STO.A007 := NOT 1;
END_REGION

REGION Network 11: Storing A008: Antivries alarm
   #STO.A008 := NOT 1;
END_REGION

REGION Network 12: Storing A009: Filter vuil verse lucht
   #STO.A009 := NOT 1;
END_REGION

REGION Network 13: Storing A010: Filter vuil extractie lucht
   #STO.A010 := NOT 1;
END_REGION

REGION Network 14: Melding M001: De pulsie ventilator is afgekoppeld via de werkschakelaar
   #STO.M001 := NOT 1;
END_REGION

REGION Network 15: Melding M002: De extractie ventilator is afgekoppeld via de werkschakelaar
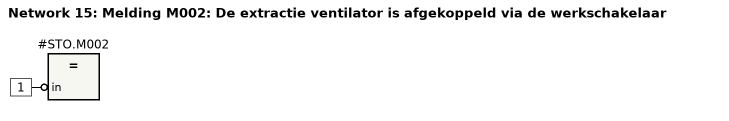
   #STO.M002 := NOT 1;
END_REGION

REGION Network 16: +++ Regelingen +++
   // PID regelingen voor luchtdebiet en temperatuur.
END_REGION

REGION Network 17: +++ Sturingen +++
   // aansturingen bepaalt door de uitgangen van de PID regelaars.
END_REGION

REGION Network 18 (SCL): EINDE
   // Variabelen van intern scada rakvlak naar outputs copieren
   #VAR_IF_LBS.WRE := #VAR.WRE;
   #VAR_IF_LBS.BMO_HAND := #VAR.BMO_HAND;
   #VAR_IF_LBS."Vrijgave pomp verwarmingsbat" := #VAR."Vrijgave pomp verwarmingsbat";
   #VAR_IF_LBS.REQ_VE := #VAR.REQ_VE;
   #VAR_IF_LBS.REQ_KO := #VAR.REQ_KO;
   #VAR_IF_LBS.STO := #STO;
END_REGION
END_FUNCTION_BLOCK

FUNCTION_BLOCK "TYPIC_C701_IF_VAT"   // FB69, FBD
TITLE = TYPIC_C701_IF_VAT: Expansievaten
{ S7_Optimized_Access := 'TRUE' }
AUTHOR : OCOTECH
FAMILY : Typical
NAME : C701.713
// Logisch Object Besturing: C701.713
// 
// De interne functie Expansievaten verzorgt de bewaking van een expansievat behorend tot de klimaatinstallatie.
// In zowel de collector verwarming als koeling is er een expansievat.
// stored: MemoryReserve 10, SetENOAutomatically false
   VAR_INPUT
      IN_AL_VE { ExternalAccessible := 'False'; ExternalVisible := 'False'; ExternalWritable := 'False'} : Bool;   // Alarm lage druk expansievat verwarming (1 = Alarm)
      IN_DME_VE { ExternalAccessible := 'False'; ExternalVisible := 'False'; ExternalWritable := 'False'} : Real;   // Drukmeting expansievat verwarming
      IN_AL_KO { ExternalAccessible := 'False'; ExternalVisible := 'False'; ExternalWritable := 'False'} : Bool;   // Alarm lage druk expansievat koeling (1 = Alarm)
      IN_DME_KO { ExternalAccessible := 'False'; ExternalVisible := 'False'; ExternalWritable := 'False'} : Real;   // Drukmeting expansievat koeling
   END_VAR
   VAR_OUTPUT
      VAR_IF_VAT { ExternalAccessible := 'False'; ExternalVisible := 'False'; ExternalWritable := 'False'} : "C701_VAR_IF_VAT_TYPIC";   // Struct met alle variabelen naar bovenliggende functies
   END_VAR
   VAR
      STO { ExternalWritable := 'False'} : Struct   // Storingen
         A001 : Bool;   // Alarm lage druk expansievat verwarming
         A002 : Bool;   // Fout drukmeting expansievat verwarming
         A003 : Bool;   // Alarm lage druk expansievat koeling
         A004 : Bool;   // Fout drukmeting expansievat koeling
      END_STRUCT;
      VAR { ExternalWritable := 'False'} : Struct   // Variabelen
         DME_VE : Real;   // Drukmeting expansievat verwarming
         DME_KO : Real;   // Drukmeting expansievat koeling
      END_STRUCT;
   END_VAR
BEGIN

REGION Network 1: START
END_REGION

REGION Network 2: +++ Metingen +++
   // inlezen van drukmeting.
END_REGION

REGION Network 3: +++ Storingen en meldingen +++
   // aanmaken van storingen en meldingen.
END_REGION

REGION Network 4: Storing A001: Alarm lage druk expansievat verwarming
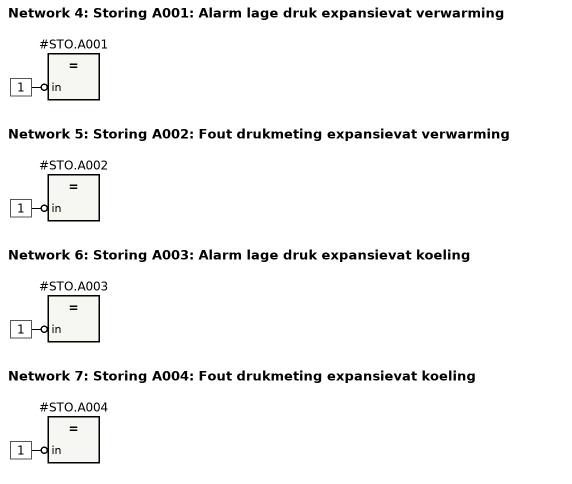
   #STO.A001 := NOT 1;
END_REGION

REGION Network 5: Storing A002: Fout drukmeting expansievat verwarming
   #STO.A002 := NOT 1;
END_REGION

REGION Network 6: Storing A003: Alarm lage druk expansievat koeling
   #STO.A003 := NOT 1;
END_REGION

REGION Network 7: Storing A004: Fout drukmeting expansievat koeling
   #STO.A004 := NOT 1;
END_REGION

REGION Network 8 (SCL): EINDE
   // Variabelen van intern scada rakvlak naar outputs copieren
   #VAR_IF_VAT.STO := #STO;
END_REGION
END_FUNCTION_BLOCK

FUNCTION_BLOCK "TYPIC_C701_IF_VAT_BUF"   // FB70, FBD
TITLE = TYPIC_C701_IF_VAT_BUF: Buffervat warm water
{ S7_Optimized_Access := 'TRUE' }
AUTHOR : OCOTECH
FAMILY : Typical
NAME : C701.714
// Logisch Object Besturing: C701.714
// 
// De interne functie Buffervat verzorgt de interne besturing, bewaking en fysieke aansturing van het buffervat behorend tot de klimaatinstallatie.
// stored: MemoryReserve 10, SetENOAutomatically false
   VAR_INPUT
      STU_IF_VAT_BUF { ExternalAccessible := 'False'; ExternalVisible := 'False'; ExternalWritable := 'False'} : Bool;   // Sturing van de interne functie klimaatregeling (IF), vrijgave door storing warmtepomp
      IN_STO { ExternalAccessible := 'False'; ExternalVisible := 'False'; ExternalWritable := 'False'} : Bool;   // Storing elektrisch weerstand
      IN_TME_MWA_INV { ExternalAccessible := 'False'; ExternalVisible := 'False'; ExternalWritable := 'False'} : Real;   // Temperatuurmeting warmwater in vertrek
      IN_TME_MWA_UITV { ExternalAccessible := 'False'; ExternalVisible := 'False'; ExternalWritable := 'False'} : Real;   // Temperatuurmeting warmwater uit vertrek
      IN_TME3_MWA { ExternalAccessible := 'False'; ExternalVisible := 'False'; ExternalWritable := 'False'} : Real;   // Temperatuurmeting warmwater in retour
      IN_TME4_MWA { ExternalAccessible := 'False'; ExternalVisible := 'False'; ExternalWritable := 'False'} : Real;   // Temperatuurmeting warmwater uit retour
   END_VAR
   VAR_OUTPUT
      VAR_IF_VAT_BUF { ExternalAccessible := 'False'; ExternalVisible := 'False'; ExternalWritable := 'False'} : "C701_VAR_IF_VAT_BUF_TYPIC";   // Struct met alle variabelen naar bovenliggende functies
      OUT_AAN { ExternalAccessible := 'False'; ExternalVisible := 'False'; ExternalWritable := 'False'} : Bool;   // Sturing elektrische weerstand (1 = Aan)
   END_VAR
   VAR
      STO { ExternalWritable := 'False'} : Struct   // Storingen
         A001 : Bool;   // Fout temperatuurmeting in vertrek
         A002 : Bool;   // Fout temperatuurmeting uit vertrek
         A003 : Bool;   // Fout temperatuurmeting in retour
         A004 : Bool;   // Fout temperatuurmeting uit retour
      END_STRUCT;
      VAR { ExternalWritable := 'False'} : Struct   // Variabelen
         TME_IN_VERTREK : Real;   // Temperatuurmeting in
         TME_UIT_VERTREK : Real;   // Temperatuurmeting uit
         TME_IN_RETOUR : Real;   // Temperatuurmeting in
         TME_UIT_RETOUR : Real;   // Temperatuurmeting uit
         TME_SWA : Real;   // Setpunt temperatuur buffervat
      END_STRUCT;
   END_VAR
BEGIN

REGION Network 1: START
END_REGION

REGION Network 2: +++ Metingen +++
   // inlezen van ingaande en uitgaande temperatuur.
END_REGION

REGION Network 3: +++ Storingen en meldingen +++
   // aanmaken van storingen en meldingen.
END_REGION

REGION Network 4: Storing A001: Fout temperatuurmeting in vertrek
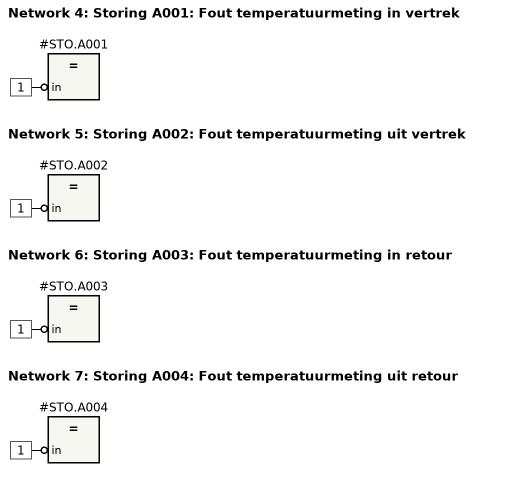
   #STO.A001 := NOT 1;
END_REGION

REGION Network 5: Storing A002: Fout temperatuurmeting uit vertrek
   #STO.A002 := NOT 1;
END_REGION

REGION Network 6: Storing A003: Fout temperatuurmeting in retour
   #STO.A003 := NOT 1;
END_REGION

REGION Network 7: Storing A004: Fout temperatuurmeting uit retour
   #STO.A004 := NOT 1;
END_REGION

REGION Network 8: +++ Sturingen +++
   // bij storing warmtepomp wordt elektrische weerstand vrijgegeven en geregeld naar setpunt.
END_REGION

REGION Network 9 (SCL): EINDE
   // Variabelen van intern scada rakvlak naar outputs copieren
   #VAR_IF_VAT_BUF.STO := #STO;
END_REGION
END_FUNCTION_BLOCK

FUNCTION_BLOCK "TYPIC_C701_IF_VEKR"   // FB96, FBD
TITLE = TYPIC_C701_IF_VEKR: Verwarmingskring
{ S7_Optimized_Access := 'TRUE' }
AUTHOR : OCOTECH
FAMILY : Typical
NAME : C701.711
// Logisch Object Besturing: C701.711
// 
// 								De interne functie Verwarmingskring verzorgt de interne besturing,
// 								bewaking en fysieke aansturing van een collectorkring behorend tot
// 								de klimaatinstallatie.
// 								Er wordt een vrijgave aan de pompen gegeven als er een warmtevraag
// 								is. De drukregeling gebeurt door de pomp zelf. Antioblokkeer
// 								beveiliging is ook instelbaar op de pomp zelf.
// 								De collector verwarming bestaat uit 2 kringen:
// 								Kring verwarmingsbatterijen
// 								Kring ventiloconvectoren en klimaatkasten
// stored: MemoryReserve 10, SetENOAutomatically false
   VAR_INPUT
      STU_IF_VEKR { ExternalAccessible := 'False'; ExternalVisible := 'False'; ExternalWritable := 'False'} : Bool;   // Sturing van de interne functie klimaatregeling (IF), warmtevraag voor kring
      IN_AAN_PMP { ExternalAccessible := 'False'; ExternalVisible := 'False'; ExternalWritable := 'False'} : Bool;   // Terugmelding aansturing pomp (1 = Aan)
      IN_THM { ExternalAccessible := 'False'; ExternalVisible := 'False'; ExternalWritable := 'False'} : Bool;   // Status thermische beveiliging (1 = OK)
      IN_DME { ExternalAccessible := 'False'; ExternalVisible := 'False'; ExternalWritable := 'False'} : Real;   // Drukmeting
      IN_TME_IN { ExternalAccessible := 'False'; ExternalVisible := 'False'; ExternalWritable := 'False'} : Real;   // Temperatuur vertrek
      IN_TME_UIT { ExternalAccessible := 'False'; ExternalVisible := 'False'; ExternalWritable := 'False'} : Real;   // Temperatuur retour
      CFG_TYD_FB { ExternalAccessible := 'False'; ExternalVisible := 'False'; ExternalWritable := 'False'} : Time;   // Vertragingstijd storing foute terugmelding
   END_VAR
   VAR_OUTPUT
      VAR_IF_VEKR { ExternalAccessible := 'False'; ExternalVisible := 'False'; ExternalWritable := 'False'} : "C701_VAR_IF_VEKR_TYPIC";   // Struct met alle variabelen naar bovenliggende functies
      OUT_VGV { ExternalAccessible := 'False'; ExternalVisible := 'False'; ExternalWritable := 'False'} : Bool;   // Vrijgave pomp
   END_VAR
   VAR_IN_OUT
      STU_VGV_VEKR_AAN : Bool;   // Vrijgave inschakelen NIET NODIG?
   END_VAR
   VAR
      STO { ExternalWritable := 'False'} : Struct   // Storingen
         A001 : Bool;   // Storing van de motorbeveiliging van de pomp
         A002 : Bool;   // Fout temperatuurmeting vertrek
         A003 : Bool;   // Fout temperatuurmeting retour
         A004 : Bool;   // Fout drukmeting
         M001 : Bool;   // De motor is afgekoppeld via de werkschakelaar
      END_STRUCT;
      VAR { ExternalWritable := 'False'} : Struct   // Variabelen
         TME_IN : Real;   // Temperatuur vertrek
         TME_UIT : Real;   // Temperatuur retour
         DME : Real;   // Druk vertrek
         VGV : Bool;   // Vrijgave voor pomp
         TYD_TOT_AAN : LInt;   // Totaal aantal draaiuren (in seconden)
         TYD_TOT_AAN_UUR : LInt;   // Totaal aantal draaiuren (in uren)
      END_STRUCT;
   END_VAR
BEGIN

REGION Network 1: START
END_REGION

REGION Network 2: +++ Metingen +++
   // inlezen van vertrek- en retourtemperatuur.
END_REGION

REGION Network 3: +++ Storingen en meldingen +++
   // aanmaken van storingen en meldingen.
END_REGION

REGION Network 4: Storing A001: Storing van de motorbeveiliging van de pomp
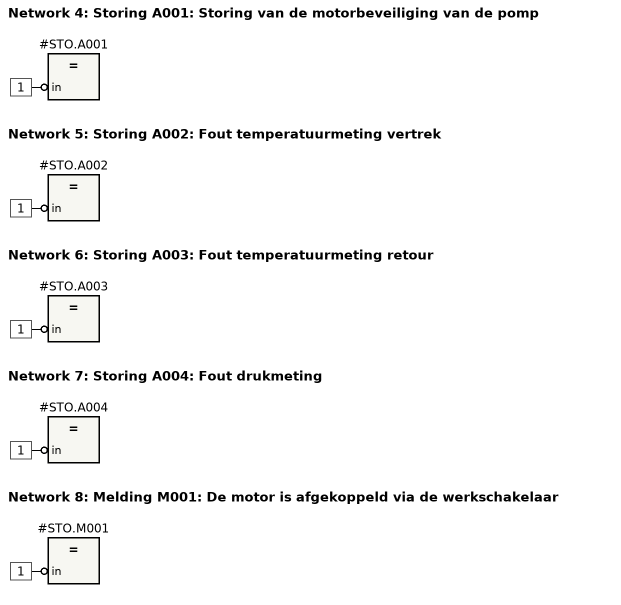
   #STO.A001 := NOT 1;
END_REGION

REGION Network 5: Storing A002: Fout temperatuurmeting vertrek
   #STO.A002 := NOT 1;
END_REGION

REGION Network 6: Storing A003: Fout temperatuurmeting retour
   #STO.A003 := NOT 1;
END_REGION

REGION Network 7: Storing A004: Fout drukmeting
   #STO.A004 := NOT 1;
END_REGION

REGION Network 8: Melding M001: De motor is afgekoppeld via de werkschakelaar
   #STO.M001 := NOT 1;
END_REGION

REGION Network 9: +++ Sturingen pomp +++
   // bij warmtevraag pomp vrijgave geven.
END_REGION

REGION Network 10: +++ Urentellers +++
   // tellen van de tijdsduur dat de motor draait.
END_REGION

REGION Network 11 (SCL): EINDE
   // Variabelen van intern scada rakvlak naar outputs copieren
   #VAR_IF_VEKR.STO := #STO;
END_REGION
END_FUNCTION_BLOCK

FUNCTION_BLOCK "TYPIC_C104_BF_NSI"   // FB95, FBD
TITLE = TYPIC_C104_BF_NSI: Noodstroominstallatie
{ S7_Optimized_Access := 'TRUE' }
AUTHOR : OCOTECH
FAMILY : Typical
NAME : C104.801
// Logisch Object Besturing: C104.801
// 
// Het doel van de BF NSI (noodstroominstallatie) is om de algemene opvolging te voorzien van de noodstroominstallatie.
// stored: MemoryReserve 10, SetENOAutomatically false
   VAR_INPUT
      STU_ALG_LCK_SIG { ExternalAccessible := 'False'; ExternalVisible := 'False'; ExternalWritable := 'False'} : USInt;   // Onderdruk alarmen
   END_VAR
   VAR_OUTPUT
      VAR_ENE_TOT_NSI { ExternalAccessible := 'False'; ExternalVisible := 'False'; ExternalWritable := 'False'} : Real;   // Totaal energieverbruik noodstroominstallatie
      VAR_VGV_NSI { ExternalAccessible := 'False'; ExternalVisible := 'False'; ExternalWritable := 'False'} : USInt;   // Vrijgave: alle noodstroomaggregaten lopen synchroon
   END_VAR
   VAR_IN_OUT
      VAR_IF_NSI : "C104_VAR_IF_NSI_TYPIC";   // Struct met alle variabelen ontvangen van de interne besturing (PMS) van de noodstroominstallatie
   END_VAR
   VAR
      SIG { ExternalWritable := 'False'} : Struct   // Signaleringen
         AB01 : Bool;   // Noodstroominstallatie niet beschikbaar
         AB02 : Bool;   // Noodstroominstallatie beperkt beschikbaar
      END_STRUCT;
      VAR { ExternalWritable := 'False'} : Struct   // Variabelen
         BSC : USInt;   // Geeft de beschikbaarheid van de noodstroominstallatie aan
         VGV_SIG_VOP : Bool;   // TRUE = Signaleringen vrijgegeven voor verkeersoperator FALSE = Onderdrukt
      END_STRUCT;
   END_VAR
BEGIN

REGION Network 1: START
END_REGION

REGION Network 2: +++ Bepalen beschikbaarheidsstatus +++
   // Beschikbaarheidsstatus (beschikbaar / beperkt beschikbaar / niet beschikbaar) bepalen.
END_REGION

REGION Network 3 (SCL): Beschikbaarheidsstatus bepalen
   IF 
       //voorwaarden "Niet beschikbaar"
       TRUE
   THEN
       //Beschikbaarheidsstatus = Niet Beschikbaar
       #VAR.BSC:= "NietBeschikbaar";
   ELSIF
       //voorwaarden "Beperkt beschikbaar"
       TRUE
   THEN
       //Beschikbaarheidsstatus = Beperkt Beschikbaar
       #VAR.BSC:= "Beperkt";
   ELSE
       //Beschikbaarheidsstatus = Beschikbaar
       #VAR.BSC:= "Beschikbaar";
   END_IF;
END_REGION

REGION Network 4: +++ Doorkoppeling totale energieverbruik HSI +++
   // Het ontvangen energieverbruik ter beschikking stellen.
END_REGION

REGION Network 5: +++ Signaleringen +++
   // Aanmaken signaleringen.
END_REGION

REGION Network 6: Signalering AB01 : Niet Beschikbaar
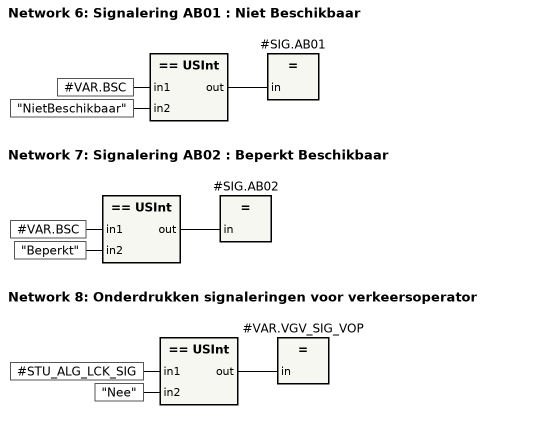
   #SIG.AB01 := #VAR.BSC = "NietBeschikbaar";
END_REGION

REGION Network 7: Signalering AB02 : Beperkt Beschikbaar
   #SIG.AB02 := #VAR.BSC = "Beperkt";
END_REGION

REGION Network 8: Onderdrukken signaleringen voor verkeersoperator
   // Via de variabele VGV_SIG_VOP wordt aan IRIS SCADA doorgegeven of signaleringen (bestemd voor de verkeersoperator) van de deze functie zichtbaar (of onderdrukt) moeten zijn.
   #VAR.VGV_SIG_VOP := #STU_ALG_LCK_SIG = "Nee";
END_REGION

REGION Network 9: EINDE
   // Variabelen van intern scada rakvlak naar outputs copieren
END_REGION
END_FUNCTION_BLOCK

FUNCTION_BLOCK "TYPIC_C104_IF_KLP"   // FB94, FBD
TITLE = TYPIC_C104_IF_KLP: Brandstofklep
{ S7_Optimized_Access := 'TRUE' }
AUTHOR : OCOTECH
FAMILY : Typical
NAME : C104.705
// Logisch Object Besturing: C104.705
// 
// De interne functie Brandstofklep verzorgt de bewaking van een brandstofklep van een noodstroomaggregaat.
// stored: MemoryReserve 10, SetENOAutomatically false
   VAR_INPUT
      EXT_AUT { ExternalAccessible := 'False'; ExternalVisible := 'False'; ExternalWritable := 'False'} : Bool;   // Externe (hoofd) beveiliging (1 = OK)
      EXT_HW { ExternalAccessible := 'False'; ExternalVisible := 'False'; ExternalWritable := 'False'} : Bool;   // Sturings hardware (PLC) bewaking (1 = OK)
      IN_STO_NOK { ExternalAccessible := 'False'; ExternalVisible := 'False'; ExternalWritable := 'False'} : Bool;   // Storing aanwezig die niet observeerbaar tot gevolg heeft
      IN_STO_OK { ExternalAccessible := 'False'; ExternalVisible := 'False'; ExternalWritable := 'False'} : Bool;   // Storing aanwezig die observeerbaarheid niet beinvloed
      IN_OPEN { ExternalAccessible := 'False'; ExternalVisible := 'False'; ExternalWritable := 'False'} : Bool;   // Brandstofklep open
      IN_TOE { ExternalAccessible := 'False'; ExternalVisible := 'False'; ExternalWritable := 'False'} : Bool;   // Brandstofklep dicht
      IN_AUT_C104 { ExternalAccessible := 'False'; ExternalVisible := 'False'; ExternalWritable := 'False'} : Bool;   // Beveiligingen: serie geschakelde terugmelding (1 = OK)
   END_VAR
   VAR_OUTPUT
      VAR_IF_KLP { ExternalAccessible := 'False'; ExternalVisible := 'False'; ExternalWritable := 'False'} : "C104_VAR_IF_KLP_TYPIC";   // Struct met alle variabelen naar bovenliggende functies
   END_VAR
   VAR
      STO { ExternalWritable := 'False'} : Struct   // Storingen
         A001 : Bool;   // Beveiliging aangesproken
         A002 : Bool;   // Brandstofklep in storing
         A003 : Bool;   // Algemene storing brandstofklep
      END_STRUCT;
      VAR { ExternalWritable := 'False'} : Struct   // Variabelen
         OPEN { ExternalAccessible := 'False'; ExternalVisible := 'False'} : Bool;   // Brandstofklep open
         TOE { ExternalAccessible := 'False'; ExternalVisible := 'False'} : Bool;   // Brandstofklep dicht
         EXT_AUT { ExternalAccessible := 'False'; ExternalVisible := 'False'} : Bool;   // Externe (hoofd) beveiliging aangesproken
         EXT_HW { ExternalAccessible := 'False'; ExternalVisible := 'False'} : Bool;   // Sturings hardware (PLC) in storing
      END_STRUCT;
   END_VAR
BEGIN

REGION Network 1: START
END_REGION

REGION Network 2: +++ Verwerking statussen +++
   // Bepalen van de statussen van de brandstofklep.
END_REGION

REGION Network 3: +++ Storingen +++
   // Verwerken van de storingsmeldingen (inputs).
END_REGION

REGION Network 4: Storing A001: Beveiliging aangesproken
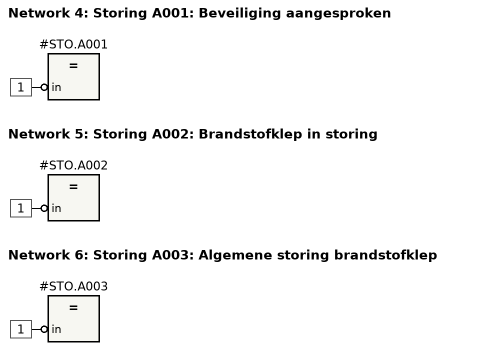
   #STO.A001 := NOT 1;
END_REGION

REGION Network 5: Storing A002: Brandstofklep in storing
   #STO.A002 := NOT 1;
END_REGION

REGION Network 6: Storing A003: Algemene storing brandstofklep
   #STO.A003 := NOT 1;
END_REGION

REGION Network 7 (SCL): EINDE
   // Variabelen van intern scada rakvlak naar outputs copieren
   #VAR_IF_KLP.OPEN := #VAR.OPEN;
   #VAR_IF_KLP.TOE := #VAR.TOE;
   #VAR_IF_KLP.EXT_AUT := #VAR.EXT_AUT;
   #VAR_IF_KLP.EXT_HW := #VAR.EXT_HW;
   #VAR_IF_KLP.STO := #STO;
END_REGION
END_FUNCTION_BLOCK

FUNCTION_BLOCK "TYPIC_C104_IF_LBS"   // FB93, FBD
TITLE = TYPIC_C104_IF_LBS: Luchtbehandelingssysteem
{ S7_Optimized_Access := 'TRUE' }
AUTHOR : OCOTECH
FAMILY : Typical
NAME : C104.704
// Logisch Object Besturing: C104.704
// 
// De interne functie Luchtbehandelingssysteem verzorgt de bewaking van het luchtbehandelingssysteem van een noodstroomaggregaat.
// stored: MemoryReserve 10, SetENOAutomatically false
   VAR_INPUT
      EXT_AUT { ExternalAccessible := 'False'; ExternalVisible := 'False'; ExternalWritable := 'False'} : Bool;   // Externe (hoofd) beveiliging (1 = OK)
      EXT_HW { ExternalAccessible := 'False'; ExternalVisible := 'False'; ExternalWritable := 'False'} : Bool;   // Sturings hardware (PLC) bewaking (1 = OK)
      IN_STO_NOK { ExternalAccessible := 'False'; ExternalVisible := 'False'; ExternalWritable := 'False'} : Bool;   // Storing aanwezig die niet observeerbaar tot gevolg heeft
      IN_STO_OK { ExternalAccessible := 'False'; ExternalVisible := 'False'; ExternalWritable := 'False'} : Bool;   // Storing aanwezig die observeerbaarheid niet beinvloed
      IN_KLP_OPEN { ExternalAccessible := 'False'; ExternalVisible := 'False'; ExternalWritable := 'False'} : Bool;   // Kleppenregister open
      IN_KLP_TOE { ExternalAccessible := 'False'; ExternalVisible := 'False'; ExternalWritable := 'False'} : Bool;   // Kleppenregister dicht
      IN_VEN_AAN { ExternalAccessible := 'False'; ExternalVisible := 'False'; ExternalWritable := 'False'} : Bool;   // Ventilator aan
      IN_AUT_C104 { ExternalAccessible := 'False'; ExternalVisible := 'False'; ExternalWritable := 'False'} : Bool;   // Beveiligingen: serie geschakelde terugmelding (1 = OK)
   END_VAR
   VAR_OUTPUT
      VAR_IF_OPT { ExternalAccessible := 'False'; ExternalVisible := 'False'; ExternalWritable := 'False'} : "C104_VAR_IF_OPT_TYPIC";   // Struct met alle variabelen naar bovenliggende functies
   END_VAR
   VAR
      STO { ExternalWritable := 'False'} : Struct   // Storingen
         A001 : Bool;   // Beveiliging aangesproken
         A002 : Bool;   // Luchtbehandelingssysteem in storing
         A003 : Bool;   // Algemene storing luchtbehandelingssysteem
      END_STRUCT;
      VAR { ExternalWritable := 'False'} : Struct   // Variabelen
         KLP_OPEN { ExternalAccessible := 'False'; ExternalVisible := 'False'} : Bool;   // Kleppenregister open
         KLP_TOE { ExternalAccessible := 'False'; ExternalVisible := 'False'} : Bool;   // Kleppenregister dicht
         VEN_AAN { ExternalAccessible := 'False'; ExternalVisible := 'False'} : Bool;   // Ventilator aan
         EXT_AUT { ExternalAccessible := 'False'; ExternalVisible := 'False'} : Bool;   // Externe (hoofd) beveiliging aangesproken
         EXT_HW { ExternalAccessible := 'False'; ExternalVisible := 'False'} : Bool;   // Sturings hardware (PLC) in storing
      END_STRUCT;
   END_VAR
BEGIN

REGION Network 1: START
END_REGION

REGION Network 2: +++ Verwerking statussen +++
   // Bepalen van de statussen van het luchtbehandelingssysteem.
END_REGION

REGION Network 3: +++ Storingen +++
   // Verwerken van de storingsmeldingen (inputs).
END_REGION

REGION Network 4: Storing A001: Beveiliging aangesproken
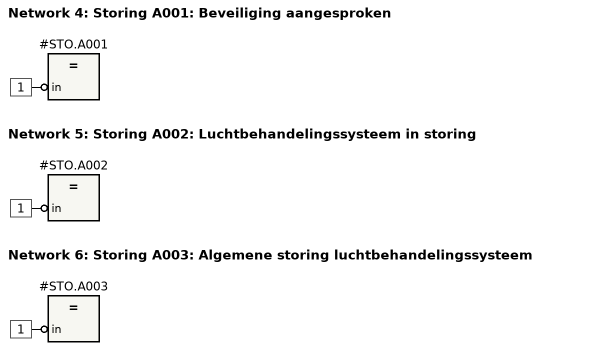
   #STO.A001 := NOT 1;
END_REGION

REGION Network 5: Storing A002: Luchtbehandelingssysteem in storing
   #STO.A002 := NOT 1;
END_REGION

REGION Network 6: Storing A003: Algemene storing luchtbehandelingssysteem
   #STO.A003 := NOT 1;
END_REGION

REGION Network 7 (SCL): EINDE
   // Variabelen van intern scada rakvlak naar outputs copieren
   #VAR_IF_OPT.KLP_OPEN := #VAR.KLP_OPEN;
   #VAR_IF_OPT.KLP_TOE := #VAR.KLP_TOE;
   #VAR_IF_OPT.VEN_AAN := #VAR.VEN_AAN;
   #VAR_IF_OPT.EXT_AUT := #VAR.EXT_AUT;
   #VAR_IF_OPT.EXT_HW := #VAR.EXT_HW;
   #VAR_IF_OPT.STO := #STO;
END_REGION
END_FUNCTION_BLOCK

FUNCTION_BLOCK "TYPIC_C104_IF_NSA"   // FB92, FBD
TITLE = TYPIC_C104_IF_NSA: Noodstroomaggregaat
{ S7_Optimized_Access := 'TRUE' }
AUTHOR : OCOTECH
FAMILY : Typical
NAME : C104.702
// Logisch Object Besturing: C104.702
// 
// De interne functie Noodstroomaggregaat verzorgt de bewaking van een noodstroomaggregaat.
// stored: MemoryReserve 10, SetENOAutomatically false
   VAR_INPUT
      EXT_AUT { ExternalAccessible := 'False'; ExternalVisible := 'False'; ExternalWritable := 'False'} : Bool;   // Externe (hoofd) beveiliging (1 = OK)
      EXT_HW { ExternalAccessible := 'False'; ExternalVisible := 'False'; ExternalWritable := 'False'} : Bool;   // Sturings hardware (PLC) bewaking (1 = OK)
      IN_STO_NOK { ExternalAccessible := 'False'; ExternalVisible := 'False'; ExternalWritable := 'False'} : Bool;   // Storing aanwezig die niet observeerbaar tot gevolg heeft
      IN_STO_OK { ExternalAccessible := 'False'; ExternalVisible := 'False'; ExternalWritable := 'False'} : Bool;   // Storing aanwezig die observeerbaarheid niet beinvloed
      IN_ENE { ExternalAccessible := 'False'; ExternalVisible := 'False'; ExternalWritable := 'False'} : Real;   // Geleverde energie per aggregaat
      IN_PHI { ExternalAccessible := 'False'; ExternalVisible := 'False'; ExternalWritable := 'False'} : Real;   // Fasehoek (cos phi)
      IN_SPA1 { ExternalAccessible := 'False'; ExternalVisible := 'False'; ExternalWritable := 'False'} : Real;   // Spanningsniveau lijn 1
      IN_SPA2 { ExternalAccessible := 'False'; ExternalVisible := 'False'; ExternalWritable := 'False'} : Real;   // Spanningsniveau lijn 2
      IN_SPA3 { ExternalAccessible := 'False'; ExternalVisible := 'False'; ExternalWritable := 'False'} : Real;   // Spanningsniveau lijn 3
      IN_STR { ExternalAccessible := 'False'; ExternalVisible := 'False'; ExternalWritable := 'False'} : Real;   // Stroomsterkte
      IN_WRE { ExternalAccessible := 'False'; ExternalVisible := 'False'; ExternalWritable := 'False'} : Bool;   // TRUE = werkingsregime: Belast FALSE = werkingsregime: Onbelast
      IN_STS1 { ExternalAccessible := 'False'; ExternalVisible := 'False'; ExternalWritable := 'False'} : Bool;   // Status: Standby
      IN_STS2 { ExternalAccessible := 'False'; ExternalVisible := 'False'; ExternalWritable := 'False'} : Bool;   // Status: Storing
      IN_STS3 { ExternalAccessible := 'False'; ExternalVisible := 'False'; ExternalWritable := 'False'} : Bool;   // Status: Uitgeschakeld
      IN_STS4 { ExternalAccessible := 'False'; ExternalVisible := 'False'; ExternalWritable := 'False'} : Bool;   // Status: Test
      IN_STS_AAN { ExternalAccessible := 'False'; ExternalVisible := 'False'; ExternalWritable := 'False'} : Bool;   // In bedrijf (Aan)
      IN_LDE { ExternalAccessible := 'False'; ExternalVisible := 'False'; ExternalWritable := 'False'} : Bool;   // Lekdetectie NSA
      IN_TYD_TOT_AAN_UUR { ExternalAccessible := 'False'; ExternalVisible := 'False'; ExternalWritable := 'False'} : LInt;   // TYD_TOT_AAN_UUR
      IN_SNS { ExternalAccessible := 'False'; ExternalVisible := 'False'; ExternalWritable := 'False'} : Bool;   // Noodstop (1 = gedeactiveerd)
      IN_OPT_LDE { ExternalAccessible := 'False'; ExternalVisible := 'False'; ExternalWritable := 'False'} : Bool;   // Lekdetectie brandstof dagtank
      IN_OPT_NIV { ExternalAccessible := 'False'; ExternalVisible := 'False'; ExternalWritable := 'False'} : Real;   // Brandstof niveau brandstof dagtank
      IN_OPT_HOOG { ExternalAccessible := 'False'; ExternalVisible := 'False'; ExternalWritable := 'False'} : Bool;   // Overvulbeveiliging brandstof dagtank aangesproken
      IN_OPT_STO { ExternalAccessible := 'False'; ExternalVisible := 'False'; ExternalWritable := 'False'} : Bool;   // Dagtank noodstroomaggregaat in storing
      IN_AUT_C104 { ExternalAccessible := 'False'; ExternalVisible := 'False'; ExternalWritable := 'False'} : Bool;   // Beveiligingen: serie geschakelde terugmelding (1 = OK)
   END_VAR
   VAR_OUTPUT
      VAR_IF_NSA { ExternalAccessible := 'False'; ExternalVisible := 'False'; ExternalWritable := 'False'} : "C104_VAR_IF_NSA_TYPIC";   // Struct met alle variabelen naar bovenliggende functies
   END_VAR
   VAR
      STO { ExternalWritable := 'False'} : Struct   // Storingen
         A001 : Bool;   // Beveiliging aangesproken
         A002 : Bool;   // Noodstroomaggregaat in storing
         A003 : Bool;   // Algemene storing noodstroomaggregaat
         A004 : Bool;   // Lekdetectie NSA
         A005 : Bool;   // Noodstop van het noodstroomaggregaat is geactiveerd
         A006 : Bool;   // Dagtank noodstroomaggregaat in storing
         A007 : Bool;   // Lekdetectie brandstof dagtank
         A008 : Bool;   // Overvulbeveiliging brandstof dagtank aangesproken
      END_STRUCT;
      VAR { ExternalWritable := 'False'} : Struct   // Variabelen
         ENE { ExternalAccessible := 'False'; ExternalVisible := 'False'} : Real;   // Geleverde energie per aggregaat [kWh]
         PHI { ExternalAccessible := 'False'; ExternalVisible := 'False'} : Real;   // Fasehoek (cos phi)
         SPA1 { ExternalAccessible := 'False'; ExternalVisible := 'False'} : Real;   // Spanningsniveau lijn 1
         SPA2 { ExternalAccessible := 'False'; ExternalVisible := 'False'} : Real;   // Spanningsniveau lijn 2
         SPA3 { ExternalAccessible := 'False'; ExternalVisible := 'False'} : Real;   // Spanningsniveau lijn 3
         STR { ExternalAccessible := 'False'; ExternalVisible := 'False'} : Real;   // Stroomsterkte
         WRE { ExternalAccessible := 'False'; ExternalVisible := 'False'} : Bool;   // TRUE = werkingsregime: Belast FALSE = werkingsregime: Onbelast
         STS1 { ExternalAccessible := 'False'; ExternalVisible := 'False'} : Bool;   // Status: Standby
         STS2 { ExternalAccessible := 'False'; ExternalVisible := 'False'} : Bool;   // Status: Storing
         STS3 { ExternalAccessible := 'False'; ExternalVisible := 'False'} : Bool;   // Status: Uitgeschakeld
         STS4 { ExternalAccessible := 'False'; ExternalVisible := 'False'} : Bool;   // Status: Test
         STS_AAN { ExternalAccessible := 'False'; ExternalVisible := 'False'} : Bool;   // In bedrijf (AAN)
         LDE { ExternalAccessible := 'False'; ExternalVisible := 'False'} : Bool;   // Lekdetectie NSA
         TYD_TOT_AAN_UUR { ExternalAccessible := 'False'; ExternalVisible := 'False'} : LInt;   // TYD_TOT_AAN_UUR
         SNS { ExternalAccessible := 'False'; ExternalVisible := 'False'} : Bool;   // Noodstop (1 = gedeactiveerd)
         OPT_LDE { ExternalAccessible := 'False'; ExternalVisible := 'False'} : Bool;   // Lekdetectie brandstof dagtank
         OPT_NIV { ExternalAccessible := 'False'; ExternalVisible := 'False'} : Real;   // Brandstof niveau brandstof dagtank
         OPT_HOOG { ExternalAccessible := 'False'; ExternalVisible := 'False'} : Bool;   // Overvulbeveiliging brandstof dagtank aangesproken
         OPT_STO { ExternalAccessible := 'False'; ExternalVisible := 'False'} : Bool;   // Dagtank noodstroomaggregaat in storing
         EXT_AUT { ExternalAccessible := 'False'; ExternalVisible := 'False'} : Bool;   // Externe (hoofd) beveiliging aangesproken
         EXT_HW { ExternalAccessible := 'False'; ExternalVisible := 'False'} : Bool;   // Sturings hardware (PLC) in storing
      END_STRUCT;
   END_VAR
BEGIN

REGION Network 1: START
END_REGION

REGION Network 2: +++ Verwerking meetwaarden en statussen +++
   // De meetwaarden en statussen van het noodstroomaggregaat worden ontvangen vanuit de interne sturing.
END_REGION

REGION Network 3: +++ Storingen +++
   // Verwerken van de storingsmeldingen (inputs).
END_REGION

REGION Network 4: Storing A001: Beveiliging aangesproken
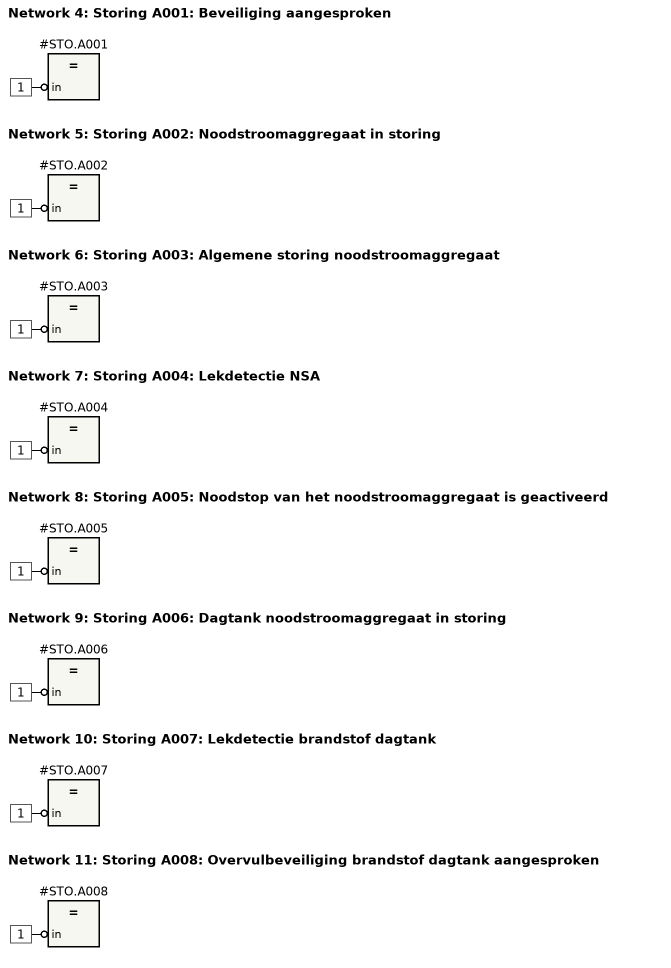
   #STO.A001 := NOT 1;
END_REGION

REGION Network 5: Storing A002: Noodstroomaggregaat in storing
   #STO.A002 := NOT 1;
END_REGION

REGION Network 6: Storing A003: Algemene storing noodstroomaggregaat
   #STO.A003 := NOT 1;
END_REGION

REGION Network 7: Storing A004: Lekdetectie NSA
   #STO.A004 := NOT 1;
END_REGION

REGION Network 8: Storing A005: Noodstop van het noodstroomaggregaat is geactiveerd
   #STO.A005 := NOT 1;
END_REGION

REGION Network 9: Storing A006: Dagtank noodstroomaggregaat in storing
   #STO.A006 := NOT 1;
END_REGION

REGION Network 10: Storing A007: Lekdetectie brandstof dagtank
   #STO.A007 := NOT 1;
END_REGION

REGION Network 11: Storing A008: Overvulbeveiliging brandstof dagtank aangesproken
   #STO.A008 := NOT 1;
END_REGION

REGION Network 12 (SCL): EINDE
   // Variabelen van intern scada rakvlak naar outputs copieren
   #VAR_IF_NSA.ENE := #VAR.ENE;
   #VAR_IF_NSA.PHI := #VAR.PHI;
   #VAR_IF_NSA.SPA1 := #VAR.SPA1;
   #VAR_IF_NSA.SPA2 := #VAR.SPA2;
   #VAR_IF_NSA.SPA3 := #VAR.SPA3;
   #VAR_IF_NSA.STR := #VAR.STR;
   #VAR_IF_NSA.WRE := #VAR.WRE;
   #VAR_IF_NSA.STS1 := #VAR.STS1;
   #VAR_IF_NSA.STS2 := #VAR.STS2;
   #VAR_IF_NSA.STS3 := #VAR.STS3;
   #VAR_IF_NSA.STS4 := #VAR.STS4;
   #VAR_IF_NSA.STS_AAN := #VAR.STS_AAN;
   #VAR_IF_NSA.LDE := #VAR.LDE;
   #VAR_IF_NSA.TYD_TOT_AAN_UUR := #VAR.TYD_TOT_AAN_UUR;
   #VAR_IF_NSA.SNS := #VAR.SNS;
   #VAR_IF_NSA.OPT_LDE := #VAR.OPT_LDE;
   #VAR_IF_NSA.OPT_NIV := #VAR.OPT_NIV;
   #VAR_IF_NSA.OPT_HOOG := #VAR.OPT_HOOG;
   #VAR_IF_NSA.OPT_STO := #VAR.OPT_STO;
   #VAR_IF_NSA.EXT_AUT := #VAR.EXT_AUT;
   #VAR_IF_NSA.EXT_HW := #VAR.EXT_HW;
   #VAR_IF_NSA.STO := #STO;
END_REGION
END_FUNCTION_BLOCK

FUNCTION_BLOCK "TYPIC_C104_IF_NSI"   // FB91, FBD
TITLE = TYPIC_C104_IF_NSI: Noodstroominstallatie
{ S7_Optimized_Access := 'TRUE' }
AUTHOR : OCOTECH
FAMILY : Typical
NAME : C104.701
// Logisch Object Besturing: C104.701
// 
// De interne functie Noodstroominstallatie verzorgt de bewaking van de noodstroominstallatie.
// stored: MemoryReserve 10, SetENOAutomatically false
   VAR_INPUT
      IN_NSI_BSC1 { ExternalAccessible := 'False'; ExternalVisible := 'False'; ExternalWritable := 'False'} : Bool;   // Noodstroominstallatie beschikbaar
      IN_NSI_BSC2 { ExternalAccessible := 'False'; ExternalVisible := 'False'; ExternalWritable := 'False'} : Bool;   // Noodstroominstallatie niet beschikbaar
      IN_NSI_BSC3 { ExternalAccessible := 'False'; ExternalVisible := 'False'; ExternalWritable := 'False'} : Bool;   // Noodstroominstallatie beperkt beschikbaar
      IN_NSI_ENE_TOT { ExternalAccessible := 'False'; ExternalVisible := 'False'; ExternalWritable := 'False'} : Real;   // Totaal energieverbruik noodstroominstallatie
      IN_AUT_C104 { ExternalAccessible := 'False'; ExternalVisible := 'False'; ExternalWritable := 'False'} : Bool;   // Beveiligingen: serie geschakelde terugmelding (1 = OK)
   END_VAR
   VAR_OUTPUT
      VAR_IF_NSI { ExternalAccessible := 'False'; ExternalVisible := 'False'; ExternalWritable := 'False'} : "C104_VAR_IF_NSI_TYPIC";   // Struct met alle variabelen naar bovenliggende functies
   END_VAR
   VAR
      VAR { ExternalWritable := 'False'} : Struct   // Variabelen
         BSC1 { ExternalAccessible := 'False'; ExternalVisible := 'False'} : Bool;   // Noodstroominstallatie beschikbaar
         BSC2 { ExternalAccessible := 'False'; ExternalVisible := 'False'} : Bool;   // Noodstroominstallatie niet beschikbaar
         BSC3 { ExternalAccessible := 'False'; ExternalVisible := 'False'} : Bool;   // Noodstroominstallatie beperkt beschikbaar
         ENE_TOT { ExternalAccessible := 'False'; ExternalVisible := 'False'} : Real;   // Totaal energieverbruik noodstroominstallatie
      END_STRUCT;
   END_VAR
BEGIN

REGION Network 1: START
END_REGION

REGION Network 2: +++ Verwerking meetwaarden en statussen +++
   // De meetwaarden en statussen van de noodstroominstallatie worden ontvangen vanuit de interne sturing.
END_REGION

REGION Network 3: +++ Storingen +++
   // Verwerken van de storingsmeldingen (inputs).
END_REGION

REGION Network 4 (SCL): EINDE
   // Variabelen van intern scada rakvlak naar outputs copieren
   #VAR_IF_NSI.BSC1 := #VAR.BSC1;
   #VAR_IF_NSI.BSC2 := #VAR.BSC2;
   #VAR_IF_NSI.BSC3 := #VAR.BSC3;
   #VAR_IF_NSI.ENE_TOT := #VAR.ENE_TOT;
END_REGION
END_FUNCTION_BLOCK

FUNCTION_BLOCK "TYPIC_C104_IF_PMP"   // FB89, FBD
TITLE = TYPIC_C104_IF_PMP: Brandstofpomp
{ S7_Optimized_Access := 'TRUE' }
AUTHOR : OCOTECH
FAMILY : Typical
NAME : C104.706
// Logisch Object Besturing: C104.706
// 
// De interne functie Brandstofpomp verzorgt de bewaking van de brandstofpomp.
// stored: MemoryReserve 10, SetENOAutomatically false
   VAR_INPUT
      EXT_AUT { ExternalAccessible := 'False'; ExternalVisible := 'False'; ExternalWritable := 'False'} : Bool;   // Externe (hoofd) beveiliging (1 = OK)
      EXT_HW { ExternalAccessible := 'False'; ExternalVisible := 'False'; ExternalWritable := 'False'} : Bool;   // Sturings hardware (PLC) bewaking (1 = OK)
      IN_STO_NOK { ExternalAccessible := 'False'; ExternalVisible := 'False'; ExternalWritable := 'False'} : Bool;   // Storing aanwezig die niet observeerbaar tot gevolg heeft
      IN_STO_OK { ExternalAccessible := 'False'; ExternalVisible := 'False'; ExternalWritable := 'False'} : Bool;   // Storing aanwezig die observeerbaarheid niet beinvloed
      IN_AAN { ExternalAccessible := 'False'; ExternalVisible := 'False'; ExternalWritable := 'False'} : Bool;   // Brandstofpomp aan
      IN_AUT_C104 { ExternalAccessible := 'False'; ExternalVisible := 'False'; ExternalWritable := 'False'} : Bool;   // Beveiligingen: serie geschakelde terugmelding (1 = OK)
   END_VAR
   VAR_OUTPUT
      VAR_IF_PMP { ExternalAccessible := 'False'; ExternalVisible := 'False'; ExternalWritable := 'False'} : "C104_VAR_IF_PMP_TYPIC";   // Struct met alle variabelen naar bovenliggende functies
   END_VAR
   VAR
      STO { ExternalWritable := 'False'} : Struct   // Storingen
         A001 : Bool;   // Beveiliging aangesproken
         A002 : Bool;   // Brandstofpomp in storing
         A003 : Bool;   // Algemene storing brandstofpomp
      END_STRUCT;
      VAR { ExternalWritable := 'False'} : Struct   // Variabelen
         AAN { ExternalAccessible := 'False'; ExternalVisible := 'False'} : Bool;   // Brandstofpomp aan
         EXT_AUT { ExternalAccessible := 'False'; ExternalVisible := 'False'} : Bool;   // Externe (hoofd) beveiliging aangesproken
         EXT_HW { ExternalAccessible := 'False'; ExternalVisible := 'False'} : Bool;   // Sturings hardware (PLC) in storing
      END_STRUCT;
   END_VAR
BEGIN

REGION Network 1: START
END_REGION

REGION Network 2: +++ Verwerking statussen +++
   // Bepalen van de statussen van het brandstofpomp.
END_REGION

REGION Network 3: +++ Storingen +++
   // Verwerken van de storingsmeldingen (inputs).
END_REGION

REGION Network 4: Storing A001: Beveiliging aangesproken
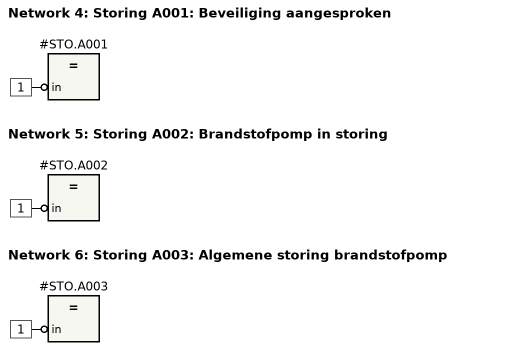
   #STO.A001 := NOT 1;
END_REGION

REGION Network 5: Storing A002: Brandstofpomp in storing
   #STO.A002 := NOT 1;
END_REGION

REGION Network 6: Storing A003: Algemene storing brandstofpomp
   #STO.A003 := NOT 1;
END_REGION

REGION Network 7 (SCL): EINDE
   // Variabelen van intern scada rakvlak naar outputs copieren
   #VAR_IF_PMP.AAN := #VAR.AAN;
   #VAR_IF_PMP.EXT_AUT := #VAR.EXT_AUT;
   #VAR_IF_PMP.EXT_HW := #VAR.EXT_HW;
   #VAR_IF_PMP.STO := #STO;
END_REGION
END_FUNCTION_BLOCK

FUNCTION_BLOCK "TYPIC_C106_BF_HSI"   // FB85, FBD
TITLE = TYPIC_C106_BF_HSI: Hoogspanningsinstallatie
{ S7_Optimized_Access := 'TRUE' }
AUTHOR : OCOTECH
FAMILY : Typical
NAME : C106.801
// Logisch Object Besturing: C106.801
// 
// Het doel van de BF HSI (hoogspanningsinstallatie) is om de algemene opvolging te voorzien van de hoogspanningsinstallatie.
// stored: MemoryReserve 10, SetENOAutomatically false
   VAR_INPUT
      STU_ALG_LCK_SIG { ExternalAccessible := 'False'; ExternalVisible := 'False'; ExternalWritable := 'False'} : USInt;   // Onderdruk alarmen
   END_VAR
   VAR_OUTPUT
      AUT_STS_HSI { ExternalAccessible := 'False'; ExternalVisible := 'False'; ExternalWritable := 'False'} : Array[0..1] of Bool;   // Standmelding van de vermogenschakelaar van de hoogspanning, naar de coordinerende functie Energiemonitor
   END_VAR
   VAR_IN_OUT
      VAR_IF_HSI : "C106_VAR_IF_HSI_TYPIC";   // Struct met alle variabelen van de interne besturing van de hoogspanningsinstallatie en de status van de hoogspanningslus
      VAR_REL : Array[*] of "C106_VAR_REL_TYPIC";   // Array met de standmelding van alle vermogenschakelaars (gekoppeld aan het beveiligingsrelais)
   END_VAR
   VAR
      SIG { ExternalWritable := 'False'} : Struct   // Signaleringen
         AB01 : Bool;   // Hoogspanningsinstallatie niet beschikbaar
         AB02 : Bool;   // Hoogspanningsinstallatie beperkt beschikbaar
         AA01 : Bool;   // Hoogspanningsinstallatie niet observeerbaar
         AA02 : Bool;   // Hoogspanningsinstallatie storing algemeen
         A001 : Bool;   // Beveiliging aangesproken
         A002 : Bool;   // Hoogspanningsinstallatie in storing
         A003 : Bool;   // Algemene storing hoogspanningsinstallatie
         A004 : Bool;   // Hoogspanningslus is geopend
      END_STRUCT;
      VAR { ExternalWritable := 'False'} : Struct   // Variabelen
         LUS_STS : USInt;   // Status van de hoogspanningslus
         BSC : USInt;   // Geeft de beschikbaarheid van de hoogspanningsinstallatie aan
         VGV_SIG_VOP : Bool;   // TRUE = Signaleringen vrijgegeven voor verkeersoperator FALSE = Onderdrukt
      END_STRUCT;
   END_VAR
BEGIN

REGION Network 1: START
END_REGION

REGION Network 2: +++ Verwerking meetwaarden en statussen +++
   // Verwerken van de ontvangen meetwaarden en statussen
END_REGION

REGION Network 3: +++ Bepalen werkingsregime hoogspanningsinstallatie +++
   // Het bepalen van het werkingsregime van de hoogspanningsinstallatie in samenspraak met de noodstroominstallatie
END_REGION

REGION Network 4: +++ Bepalen status hoogspanningslus +++
   // De status van de hoogspanningslus geeft aan of de hoogspanningslus onderbroken is of niet
END_REGION

REGION Network 5: +++ Doorkoppelen gegevens vermogen en energie naar coördinerende functie energiemonitoring +++
   // De actuele vermogen en energiemeting wordt doorgegeven aan de coordinerende functie Energievoorziening.
END_REGION

REGION Network 6: +++ Doorkoppelen status vermogenschakelaars HSI naar coördinerende functie energiemonitoring +++
   // De status van de vermogenschakelaars van de hoogspanningsinstallatie wordt doorgegeven aan de coordinerende functie Energievoorziening
END_REGION

REGION Network 7: +++ Bepalen beschikbaarheidsstatus +++
   // Beschikbaarheidsstatus (beschikbaar / beperkt beschikbaar / niet beschikbaar) bepalen.
END_REGION

REGION Network 8 (SCL): Beschikbaarheidsstatus bepalen
   IF 
       //voorwaarden "Niet beschikbaar"
       TRUE
   THEN
       //Beschikbaarheidsstatus = Niet Beschikbaar
       #VAR.BSC:= "NietBeschikbaar";
   ELSIF
       //voorwaarden "Beperkt beschikbaar"
       TRUE
   THEN
       //Beschikbaarheidsstatus = Beperkt Beschikbaar
       #VAR.BSC:= "Beperkt";
   ELSE
       //Beschikbaarheidsstatus = Beschikbaar
       #VAR.BSC:= "Beschikbaar";
   END_IF;
END_REGION

REGION Network 9: +++ Signaleringen +++
   // Aanmaken signaleringen
END_REGION

REGION Network 10 (SCL): Signaleringen voor de onderhoudsoperator
   // Signalering van de storingen ontvangen vanuit de interne sturing
   #SIG.A001 := #VAR_IF_HSI.STO.A001;
   #SIG.A002 := #VAR_IF_HSI.STO.A002;
   #SIG.A003 := #VAR_IF_HSI.STO.A003;
   #SIG.A004 := #VAR_IF_HSI.STO.A004;
END_REGION

REGION Network 11: Signalering AB01 : Niet Beschikbaar
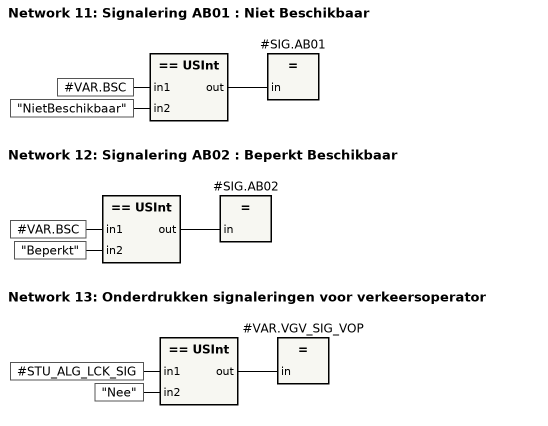
   #SIG.AB01 := #VAR.BSC = "NietBeschikbaar";
END_REGION

REGION Network 12: Signalering AB02 : Beperkt Beschikbaar
   #SIG.AB02 := #VAR.BSC = "Beperkt";
END_REGION

REGION Network 13: Onderdrukken signaleringen voor verkeersoperator
   // Via de variabele VGV_SIG_VOP wordt aan IRIS SCADA doorgegeven of signaleringen (bestemd voor de verkeersoperator) van de deze functie zichtbaar (of onderdrukt) moeten zijn.
   #VAR.VGV_SIG_VOP := #STU_ALG_LCK_SIG = "Nee";
END_REGION

REGION Network 14: EINDE
   // Variabelen van intern scada rakvlak naar outputs copieren
END_REGION
END_FUNCTION_BLOCK

FUNCTION_BLOCK "TYPIC_C106_IF_HSI"   // FB99, FBD
TITLE = TYPIC_C106_IF_HSI: Hoogspanningsinstallatie
{ S7_Optimized_Access := 'TRUE' }
AUTHOR : OCOTECH
FAMILY : Typical
NAME : C106.701
// Logisch Object Besturing: C106.701
// 
// De interne functie Hoogspanningsinstallatie verzorgt de bewaking van een hoogspanningsinstallatie.
// stored: MemoryReserve 10, SetENOAutomatically false
   VAR_INPUT
      EXT_AUT { ExternalAccessible := 'False'; ExternalVisible := 'False'; ExternalWritable := 'False'} : Bool;   // Externe (hoofd) beveiliging (1 = OK)
      EXT_HW { ExternalAccessible := 'False'; ExternalVisible := 'False'; ExternalWritable := 'False'} : Bool;   // Sturings hardware (PLC) bewaking (1 = OK)
      IN_STO_NOK { ExternalAccessible := 'False'; ExternalVisible := 'False'; ExternalWritable := 'False'} : Bool;   // Storing aanwezig die niet observeerbaar tot gevolg heeft
      IN_STO_OK { ExternalAccessible := 'False'; ExternalVisible := 'False'; ExternalWritable := 'False'} : Bool;   // Storing aanwezig die observeerbaarheid niet beinvloed
      IN_HSI_BSC1 { ExternalAccessible := 'False'; ExternalVisible := 'False'; ExternalWritable := 'False'} : Bool;   // Hoogspanningsinstallatie beschikbaar
      IN_HSI_BSC2 { ExternalAccessible := 'False'; ExternalVisible := 'False'; ExternalWritable := 'False'} : Bool;   // Hoogspanningsinstallatie niet beschikbaar
      IN_HSI_BSC3 { ExternalAccessible := 'False'; ExternalVisible := 'False'; ExternalWritable := 'False'} : Bool;   // Hoogspanningsinstallatie beperkt beschikbaar
      IN_LUS_TOE { ExternalAccessible := 'False'; ExternalVisible := 'False'; ExternalWritable := 'False'} : Bool;   // Hoogspanningslus is gesloten
      IN_WRE1 { ExternalAccessible := 'False'; ExternalVisible := 'False'; ExternalWritable := 'False'} : Bool;   // Werkingsregime: Netbedrijf
      IN_WRE2 { ExternalAccessible := 'False'; ExternalVisible := 'False'; ExternalWritable := 'False'} : Bool;   // Werkingsregime: Parallelbedrijf
      IN_WRE3 { ExternalAccessible := 'False'; ExternalVisible := 'False'; ExternalWritable := 'False'} : Bool;   // Werkingsregime: Eilandbedrijf
      IN_HSI_ENE_TOT { ExternalAccessible := 'False'; ExternalVisible := 'False'; ExternalWritable := 'False'} : Real;   // Totaal energieverbruik hoogspanningsinstallatie
      IN_AUT_C106 { ExternalAccessible := 'False'; ExternalVisible := 'False'; ExternalWritable := 'False'} : Bool;   // Beveiligingen: serie geschakelde terugmelding (1 = OK)
   END_VAR
   VAR_OUTPUT
      VAR_IF_HSI { ExternalAccessible := 'False'; ExternalVisible := 'False'; ExternalWritable := 'False'} : "C106_VAR_IF_HSI_TYPIC";   // Struct met alle variabelen naar bovenliggende functies
   END_VAR
   VAR
      STO { ExternalWritable := 'False'} : Struct   // Storingen
         A001 : Bool;   // Beveiliging aangesproken
         A002 : Bool;   // Hoogspanningsinstallatie in storing
         A003 : Bool;   // Algemene storing hoogspanningsinstallatie
         A004 : Bool;   // Hoogspanningslus is geopend
      END_STRUCT;
      VAR { ExternalWritable := 'False'} : Struct   // Variabelen
         BSC1 : Bool;   // Hoogspanningsinstallatie beschikbaar
         BSC2 : Bool;   // Hoogspanningsinstallatie niet beschikbaar
         BSC3 : Bool;   // Hoogspanningsinstallatie beperkt beschikbaar
         WRE1 : Bool;   // Werkingsregime: Netbedrijf
         WRE2 : Bool;   // Werkingsregime: Parallelbedrijf
         WRE3 : Bool;   // Werkingsregime: Eilandbedrijf
         LUS_TOE : Bool;   // Hoogspanningslus is gesloten
         EXT_AUT { ExternalAccessible := 'False'; ExternalVisible := 'False'} : Bool;   // Externe (hoofd) beveiliging aangesproken
         EXT_HW { ExternalAccessible := 'False'; ExternalVisible := 'False'} : Bool;   // Sturings hardware (PLC) in storing
      END_STRUCT;
   END_VAR
BEGIN

REGION Network 1: START
END_REGION

REGION Network 2: +++ Verwerking meetwaarden en statussen +++
   // De meetwaarde en status wordt ontvangen vanuit de interne sturing.
END_REGION

REGION Network 3: +++ Storingen +++
   // Verwerken van de storingsmeldingen (inputs).
END_REGION

REGION Network 4: Storing A001: Beveiliging aangesproken
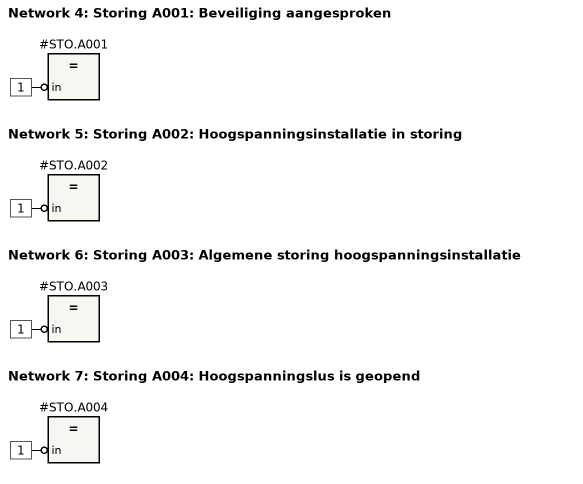
   #STO.A001 := NOT 1;
END_REGION

REGION Network 5: Storing A002: Hoogspanningsinstallatie in storing
   #STO.A002 := NOT 1;
END_REGION

REGION Network 6: Storing A003: Algemene storing hoogspanningsinstallatie
   #STO.A003 := NOT 1;
END_REGION

REGION Network 7: Storing A004: Hoogspanningslus is geopend
   #STO.A004 := NOT 1;
END_REGION

REGION Network 8 (SCL): EINDE
   // Variabelen van intern scada rakvlak naar outputs copieren
   #VAR_IF_HSI.BSC1 := #VAR.BSC1;
   #VAR_IF_HSI.BSC2 := #VAR.BSC2;
   #VAR_IF_HSI.BSC3 := #VAR.BSC3;
   #VAR_IF_HSI.WRE1 := #VAR.WRE1;
   #VAR_IF_HSI.WRE2 := #VAR.WRE2;
   #VAR_IF_HSI.WRE3 := #VAR.WRE3;
   #VAR_IF_HSI.LUS_TOE := #VAR.LUS_TOE;
   #VAR_IF_HSI.EXT_AUT := #VAR.EXT_AUT;
   #VAR_IF_HSI.EXT_HW := #VAR.EXT_HW;
   #VAR_IF_HSI.STO := #STO;
END_REGION
END_FUNCTION_BLOCK

FUNCTION_BLOCK "TYPIC_C106_IF_MVI"   // FB84, FBD
TITLE = TYPIC_C106_IF_MVI: Hoogspanningsverdeelbord
{ S7_Optimized_Access := 'TRUE' }
AUTHOR : OCOTECH
FAMILY : Typical
NAME : C106.702
// Logisch Object Besturing: C106.702
// 
// De interne functie Hoogspanningsverdeelbord verzorgt de bewaking van een oogspanningsverdeelbord.
// stored: MemoryReserve 10, SetENOAutomatically false
   VAR_INPUT
      EXT_AUT { ExternalAccessible := 'False'; ExternalVisible := 'False'; ExternalWritable := 'False'} : Bool;   // Externe (hoofd) beveiliging (1 = OK)
      EXT_HW { ExternalAccessible := 'False'; ExternalVisible := 'False'; ExternalWritable := 'False'} : Bool;   // Sturings hardware (PLC) bewaking (1 = OK)
      IN_PWR1 { ExternalAccessible := 'False'; ExternalVisible := 'False'; ExternalWritable := 'False'} : Real;   // Actief vermogen
      IN_PWR2 { ExternalAccessible := 'False'; ExternalVisible := 'False'; ExternalWritable := 'False'} : Real;   // Reactief vermogen
      IN_SPA1 { ExternalAccessible := 'False'; ExternalVisible := 'False'; ExternalWritable := 'False'} : Real;   // Lijnspanning 1
      IN_SPA2 { ExternalAccessible := 'False'; ExternalVisible := 'False'; ExternalWritable := 'False'} : Real;   // Lijnspanning 2
      IN_SPA3 { ExternalAccessible := 'False'; ExternalVisible := 'False'; ExternalWritable := 'False'} : Real;   // Lijnspanning 3
      IN_PSU_STO { ExternalAccessible := 'False'; ExternalVisible := 'False'; ExternalWritable := 'False'} : Bool;   // Storing door een fout op de UPS
      IN_PSU_AUT { ExternalAccessible := 'False'; ExternalVisible := 'False'; ExternalWritable := 'False'} : Bool;   // Verzamelalarm actief: de beveiliging van de hulpvoeding is getript
      IN_AUT_C106 { ExternalAccessible := 'False'; ExternalVisible := 'False'; ExternalWritable := 'False'} : Bool;   // Beveiligingen: serie geschakelde terugmelding (1 = OK)
   END_VAR
   VAR_OUTPUT
      VAR_IF_MVI { ExternalAccessible := 'False'; ExternalVisible := 'False'; ExternalWritable := 'False'} : "C106_VAR_IF_MVI_TYPIC";   // Struct met alle variabelen naar bovenliggende functies
   END_VAR
   VAR
      STO { ExternalWritable := 'False'} : Struct   // Storingen
         A001 : Bool;   // Beveiliging aangesproken
         A002 : Bool;   // Hoogspanningsverdeelbord in storing
         A003 : Bool;   // Algemene storing hoogspanningsverdeelbord
         A004 : Bool;   // Alarm door een fout op de UPS
         A005 : Bool;   // Verzamelalarm actief: de beveiliging van de hulpvoeding is getript
      END_STRUCT;
      VAR { ExternalWritable := 'False'} : Struct   // Variabelen
         PWR1 : Real;   // Geleverde actief vermogen per aggregaat
         PWR2 : Real;   // Geleverde reactief vermogen per aggregaat
         SPA1 : Real;   // Spanningsniveau lijn 1
         SPA2 : Real;   // Spanningsniveau lijn 2
         SPA3 : Real;   // Spanningsniveau lijn 3
         PSU_STO : Bool;   // Storing door een fout op de UPS
         PSU_AUT : Bool;   // Verzamelalarm actief: de beveiliging van de hulpvoeding is getript
         EXT_AUT { ExternalAccessible := 'False'; ExternalVisible := 'False'} : Bool;   // Externe (hoofd) beveiliging aangesproken
         EXT_HW { ExternalAccessible := 'False'; ExternalVisible := 'False'} : Bool;   // Sturings hardware (PLC) in storing
      END_STRUCT;
   END_VAR
BEGIN

REGION Network 1: START
END_REGION

REGION Network 2: +++ Verwerking meetwaarden en statussen +++
   // De meetwaarde en status wordt ontvangen vanuit de interne sturing.
END_REGION

REGION Network 3: +++ Storingen +++
   // Verwerken van de storingsmeldingen (inputs).
END_REGION

REGION Network 4: Storing A001: Beveiliging aangesproken
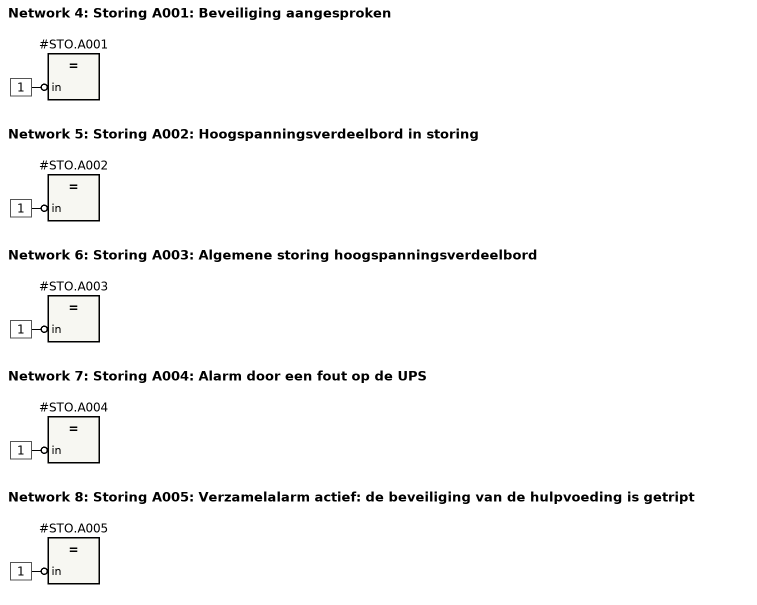
   #STO.A001 := NOT 1;
END_REGION

REGION Network 5: Storing A002: Hoogspanningsverdeelbord in storing
   #STO.A002 := NOT 1;
END_REGION

REGION Network 6: Storing A003: Algemene storing hoogspanningsverdeelbord
   #STO.A003 := NOT 1;
END_REGION

REGION Network 7: Storing A004: Alarm door een fout op de UPS
   #STO.A004 := NOT 1;
END_REGION

REGION Network 8: Storing A005: Verzamelalarm actief: de beveiliging van de hulpvoeding is getript
   #STO.A005 := NOT 1;
END_REGION

REGION Network 9 (SCL): EINDE
   // Variabelen van intern scada rakvlak naar outputs copieren
   #VAR_IF_MVI.PWR1 := #VAR.PWR1;
   #VAR_IF_MVI.PWR2 := #VAR.PWR2;
   #VAR_IF_MVI.SPA1 := #VAR.SPA1;
   #VAR_IF_MVI.SPA2 := #VAR.SPA2;
   #VAR_IF_MVI.SPA3 := #VAR.SPA3;
   #VAR_IF_MVI.PSU_STO := #VAR.PSU_STO;
   #VAR_IF_MVI.PSU_AUT := #VAR.PSU_AUT;
   #VAR_IF_MVI.EXT_AUT := #VAR.EXT_AUT;
   #VAR_IF_MVI.EXT_HW := #VAR.EXT_HW;
   #VAR_IF_MVI.STO := #STO;
END_REGION
END_FUNCTION_BLOCK

FUNCTION_BLOCK "TYPIC_C106_IF_NET"   // FB82, FBD
TITLE = TYPIC_C106_IF_NET: Netaansluiting
{ S7_Optimized_Access := 'TRUE' }
AUTHOR : OCOTECH
FAMILY : Typical
NAME : C106.705
// Logisch Object Besturing: C106.705
// 
// De interne functie netaansluiting verzorgt de bewaking van een netaansluiting.
// stored: MemoryReserve 10, SetENOAutomatically false
   VAR_INPUT
      EXT_AUT { ExternalAccessible := 'False'; ExternalVisible := 'False'; ExternalWritable := 'False'} : Bool;   // Externe (hoofd) beveiliging (1 = OK)
      EXT_HW { ExternalAccessible := 'False'; ExternalVisible := 'False'; ExternalWritable := 'False'} : Bool;   // Sturings hardware (PLC) bewaking (1 = OK)
      IN_STO_NOK { ExternalAccessible := 'False'; ExternalVisible := 'False'; ExternalWritable := 'False'} : Bool;   // Storing aanwezig die niet observeerbaar tot gevolg heeft
      IN_STO_OK { ExternalAccessible := 'False'; ExternalVisible := 'False'; ExternalWritable := 'False'} : Bool;   // Storing aanwezig die observeerbaarheid niet beinvloed
      IN_NET_BSC1 { ExternalAccessible := 'False'; ExternalVisible := 'False'; ExternalWritable := 'False'} : Bool;   // Netaansluiting beschikbaar
      IN_NET_BSC2 { ExternalAccessible := 'False'; ExternalVisible := 'False'; ExternalWritable := 'False'} : Bool;   // Netaansluiting niet beschikbaar
      IN_NET_BSC3 { ExternalAccessible := 'False'; ExternalVisible := 'False'; ExternalWritable := 'False'} : Bool;   // Netaansluiting beperkt beschikbaar
      IN_STS_KR { ExternalAccessible := 'False'; ExternalVisible := 'False'; ExternalWritable := 'False'} : Bool;   // Kritiek
      IN_STS_GKR { ExternalAccessible := 'False'; ExternalVisible := 'False'; ExternalWritable := 'False'} : Bool;   // Gestopt kritiek
      IN_TYD_GKR { ExternalAccessible := 'False'; ExternalVisible := 'False'; ExternalWritable := 'False'} : Real;   // Tijdverloop voor Gestopt Kritiek
      IN_AUT_C106 { ExternalAccessible := 'False'; ExternalVisible := 'False'; ExternalWritable := 'False'} : Bool;   // Beveiligingen: serie geschakelde terugmelding (1 = OK)
   END_VAR
   VAR_OUTPUT
      VAR_IF_NET { ExternalAccessible := 'False'; ExternalVisible := 'False'; ExternalWritable := 'False'} : "C106_VAR_IF_NET_TYPIC";   // Struct met alle variabelen naar bovenliggende functies
   END_VAR
   VAR
      STO { ExternalWritable := 'False'} : Struct   // Storingen
         A001 : Bool;   // Beveiliging aangesproken
         A002 : Bool;   // Netaansluiting in storing
         A003 : Bool;   // Algemene storing netaansluiting
         A004 : Bool;   // Geen netaansluiting beschikbaar
         A005 : Bool;   // NSA niet gestart na uitval netaansluiting
      END_STRUCT;
      VAR { ExternalWritable := 'False'} : Struct   // Variabelen
         BSC1 { ExternalAccessible := 'False'; ExternalVisible := 'False'} : Bool;   // Netaansluiting beschikbaar
         BSC2 { ExternalAccessible := 'False'; ExternalVisible := 'False'} : Bool;   // Netaansluiting niet beschikbaar
         BSC3 { ExternalAccessible := 'False'; ExternalVisible := 'False'} : Bool;   // Netaansluiting beperkt beschikbaar
         STS_KR { ExternalAccessible := 'False'; ExternalVisible := 'False'} : Bool;   // Kritiek
         STS_GKR { ExternalAccessible := 'False'; ExternalVisible := 'False'} : Bool;   // Gestopt kritiek
         TYD_GKR { ExternalAccessible := 'False'; ExternalVisible := 'False'} : Real;   // Tijdverloop voor Gestopt Kritiek
         EXT_AUT { ExternalAccessible := 'False'; ExternalVisible := 'False'} : Bool;   // Externe (hoofd) beveiliging aangesproken
         EXT_HW { ExternalAccessible := 'False'; ExternalVisible := 'False'} : Bool;   // Sturings hardware (PLC) in storing
      END_STRUCT;
   END_VAR
BEGIN

REGION Network 1: START
END_REGION

REGION Network 2: +++ Verwerking meetwaarden en statussen +++
   // De meetwaarde en status wordt ontvangen vanuit de interne sturing.
END_REGION

REGION Network 3: +++ Storingen +++
   // Verwerken van de storingsmeldingen (inputs).
END_REGION

REGION Network 4: Storing A001: Beveiliging aangesproken
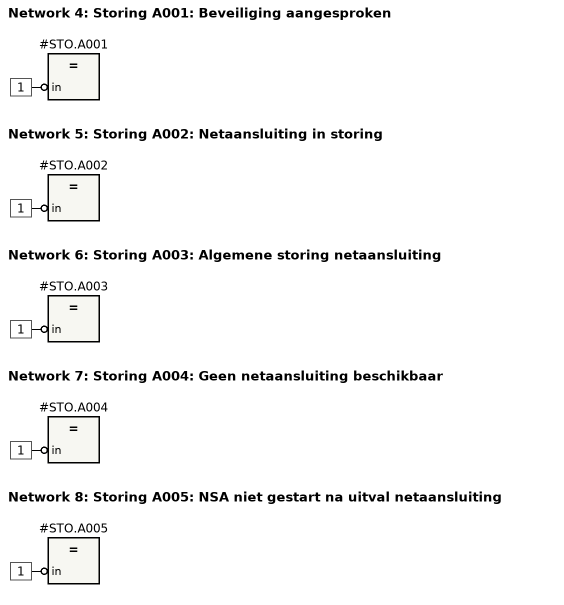
   #STO.A001 := NOT 1;
END_REGION

REGION Network 5: Storing A002: Netaansluiting in storing
   #STO.A002 := NOT 1;
END_REGION

REGION Network 6: Storing A003: Algemene storing netaansluiting
   #STO.A003 := NOT 1;
END_REGION

REGION Network 7: Storing A004: Geen netaansluiting beschikbaar
   #STO.A004 := NOT 1;
END_REGION

REGION Network 8: Storing A005: NSA niet gestart na uitval netaansluiting
   #STO.A005 := NOT 1;
END_REGION

REGION Network 9 (SCL): EINDE
   // Variabelen van intern scada rakvlak naar outputs copieren
   #VAR_IF_NET.BSC1 := #VAR.BSC1;
   #VAR_IF_NET.BSC2 := #VAR.BSC2;
   #VAR_IF_NET.BSC3 := #VAR.BSC3;
   #VAR_IF_NET.STS_KR := #VAR.STS_KR;
   #VAR_IF_NET.STS_GKR := #VAR.STS_GKR;
   #VAR_IF_NET.TYD_GKR := #VAR.TYD_GKR;
   #VAR_IF_NET.EXT_AUT := #VAR.EXT_AUT;
   #VAR_IF_NET.EXT_HW := #VAR.EXT_HW;
   #VAR_IF_NET.STO := #STO;
END_REGION
END_FUNCTION_BLOCK

FUNCTION_BLOCK "TYPIC_C106_IF_REL"   // FB81, FBD
TITLE = TYPIC_C106_IF_REL: Beveilingsrelais
{ S7_Optimized_Access := 'TRUE' }
AUTHOR : OCOTECH
FAMILY : Typical
NAME : C106.703
// Logisch Object Besturing: C106.703
// 
// De interne functie Beveiligingsrelais verzorgt de bewaking van een beveiligingsrelais.
// stored: MemoryReserve 10, SetENOAutomatically false
   VAR_INPUT
      EXT_AUT { ExternalAccessible := 'False'; ExternalVisible := 'False'; ExternalWritable := 'False'} : Bool;   // Externe (hoofd) beveiliging (1 = OK)
      EXT_HW { ExternalAccessible := 'False'; ExternalVisible := 'False'; ExternalWritable := 'False'} : Bool;   // Sturings hardware (PLC) bewaking (1 = OK)
      CFG_SYNC { ExternalAccessible := 'False'; ExternalVisible := 'False'; ExternalWritable := 'False'} : Bool;   // Type beveiligingsrelais: TRUE = Lijndifferentieel-beveiligingsrelais FALSE = Overstroom-beveiligingsrelais
      IN_STO_NOK { ExternalAccessible := 'False'; ExternalVisible := 'False'; ExternalWritable := 'False'} : Bool;   // Storing aanwezig die niet observeerbaar tot gevolg heeft
      IN_STO_OK { ExternalAccessible := 'False'; ExternalVisible := 'False'; ExternalWritable := 'False'} : Bool;   // Storing aanwezig die observeerbaarheid niet beinvloed
      IN_REL_ALM { ExternalAccessible := 'False'; ExternalVisible := 'False'; ExternalWritable := 'False'} : Bool;   // Alarm per beveiligingsrelais per uitschakelbevel: TRUE = OK / FALSE = Alarm
      IN_AUT_TOE { ExternalAccessible := 'False'; ExternalVisible := 'False'; ExternalWritable := 'False'} : Bool;   // Vermogenschakelaar TOE (gesloten)
      IN_SCA_TOE { ExternalAccessible := 'False'; ExternalVisible := 'False'; ExternalWritable := 'False'} : Bool;   // Aardingschakelaar TOE (gesloten)
      IN_SYNC { ExternalAccessible := 'False'; ExternalVisible := 'False'; ExternalWritable := 'False'} : Bool;   // Lijndifferentieel beveiligingsrelais loopt synchroon
      IN_AUT_C106 { ExternalAccessible := 'False'; ExternalVisible := 'False'; ExternalWritable := 'False'} : Bool;   // Beveiligingen: serie geschakelde terugmelding (1 = OK)
   END_VAR
   VAR_OUTPUT
      VAR_IF_REL { ExternalAccessible := 'False'; ExternalVisible := 'False'; ExternalWritable := 'False'} : "C106_VAR_IF_REL_TYPIC";   // Struct met alle variabelen naar bovenliggende functies
   END_VAR
   VAR
      STO { ExternalWritable := 'False'} : Struct   // Storingen
         A001 : Bool;   // Beveiliging aangesproken
         A002 : Bool;   // Beveiligingsrelais in storing
         A003 : Bool;   // Algemene storing beveiligingsrelais
         A004 : Bool;   // Alarm beveiligingsrelais: Uitschakelbevel
         A005 : Bool;   // Lijndifferentieel-beveiligingsrelais loopt niet synchroon met zijn tegenhanger
      END_STRUCT;
      VAR { ExternalWritable := 'False'} : Struct   // Variabelen
         ALM { ExternalAccessible := 'False'; ExternalVisible := 'False'} : Bool;   // Alarm per beveiligingsrelais per uitschakelbevel: TRUE = OK / FALSE = Alarm
         AUT_TOE { ExternalAccessible := 'False'; ExternalVisible := 'False'} : Bool;   // Vermogenschakelaar TOE (gesloten)
         SCA_TOE { ExternalAccessible := 'False'; ExternalVisible := 'False'} : Bool;   // Aardingschakelaar TOE (gesloten)
         SYNC { ExternalAccessible := 'False'; ExternalVisible := 'False'} : Bool;   // Lijndifferentieel beveiligingsrelais loopt synchroon
         EXT_AUT { ExternalAccessible := 'False'; ExternalVisible := 'False'} : Bool;   // Externe (hoofd) beveiliging aangesproken
         EXT_HW { ExternalAccessible := 'False'; ExternalVisible := 'False'} : Bool;   // Sturings hardware (PLC) in storing
      END_STRUCT;
   END_VAR
BEGIN

REGION Network 1: START
END_REGION

REGION Network 2: +++ Verwerking meetwaarden en statussen +++
   // De meetwaarde en status wordt ontvangen vanuit de interne sturing.
END_REGION

REGION Network 3: +++ Storingen +++
   // Verwerken van de storingsmeldingen (inputs).
END_REGION

REGION Network 4: Storing A001: Beveiliging aangesproken
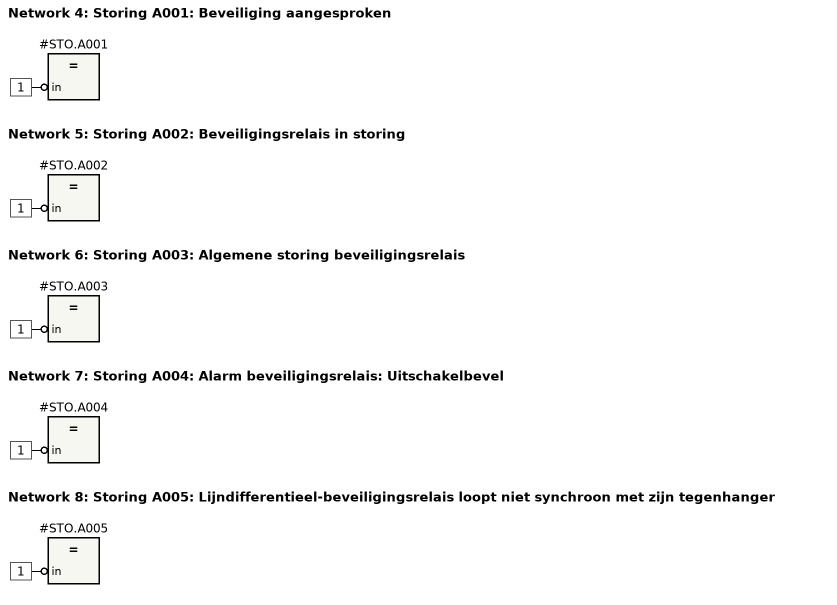
   #STO.A001 := NOT 1;
END_REGION

REGION Network 5: Storing A002: Beveiligingsrelais in storing
   #STO.A002 := NOT 1;
END_REGION

REGION Network 6: Storing A003: Algemene storing beveiligingsrelais
   #STO.A003 := NOT 1;
END_REGION

REGION Network 7: Storing A004: Alarm beveiligingsrelais: Uitschakelbevel
   #STO.A004 := NOT 1;
END_REGION

REGION Network 8: Storing A005: Lijndifferentieel-beveiligingsrelais loopt niet synchroon met zijn tegenhanger
   #STO.A005 := NOT 1;
END_REGION

REGION Network 9 (SCL): EINDE
   // Variabelen van intern scada rakvlak naar outputs copieren
   #VAR_IF_REL.ALM := #VAR.ALM;
   #VAR_IF_REL.AUT_TOE := #VAR.AUT_TOE;
   #VAR_IF_REL.SCA_TOE := #VAR.SCA_TOE;
   #VAR_IF_REL.SYNC := #VAR.SYNC;
   #VAR_IF_REL.EXT_AUT := #VAR.EXT_AUT;
   #VAR_IF_REL.EXT_HW := #VAR.EXT_HW;
END_REGION
END_FUNCTION_BLOCK

